METHOD RaiseSyncUnitEvent
VAR_INPUT
	EventId	  : UDINT;
	Argument1 : STRING := '';
	Argument2 : STRING := '';
	Argument3 : STRING := '';
END_VAR
IF Argument3 <> '' THEN
	SyncUnitEvents.Arguments(EventId).Clear().AddString(Argument1).AddString(Argument2).AddString(Argument3);
ELSIF Argument2 <> '' THEN
	SyncUnitEvents.Arguments(EventId).Clear().AddString(Argument1).AddString(Argument2);
ELSIF Argument1 <> '' THEN
	SyncUnitEvents.Arguments(EventId).Clear().AddString(Argument1);
ELSE
	SyncUnitEvents.Arguments(EventId).Clear();
END_IF

SyncUnitEvents.RaiseEvent(EventId);
END_METHOD

METHOD Reset
SyncUnitEvents.Reset();
EtherCatMasterEvents.Reset();
END_METHOD

METHOD SetEventReactions
VAR_INPUT
	Verbose	 : DINT := 0;
	Info	 : DINT := 1;
	Warning	 : DINT := 2;
	Error	 : DINT := 3;
	Critical : DINT := 4;
END_VAR
SyncUnitEvents.SetEventReactions(Verbose,
								 Info,
								 Warning,
								 Error,
								 Critical);

EtherCatMasterEvents.SetEventReactions(Verbose,
									   Info,
									   Warning,
									   Error,
									   Critical);
END_METHOD

(*FB_Init is always available implicitly and it is used primarily for initialization.
The return value is not evaluated. For a specific influence, you can also declare the
methods explicitly and provide additional code there with the standard initialization
code. You can evaluate the return value.*)
METHOD FB_Init : BOOL
VAR_INPUT
	(* TRUE: the retain variables are initialized (reset warm / reset cold)*)
	bInitRetains : BOOL;

	(* TRUE: the instance will be copied to the copy code afterward (online change)   *)
	bInCopyCode				 : BOOL;
	Name					 : Core.T_MaxString;
	EtherCatMasterDiagnostic : I_EtherCatMasterDiagnostic;
END_VAR
THIS^.EtherCatMasterDiagnostic := EtherCatMasterDiagnostic;
THIS^.EtherCatMasterDiagnostic.RegisterEventProvider(THIS^);
SyncUnitEvents.GenerateTcEvents(EtherCatMasterDiagnostic.Name, ADR(TC_Events.SyncUnit), SIZEOF(ST_SyncUnit));
EtherCatMasterEvents.GenerateTcEvents(EtherCatMasterDiagnostic.Name, ADR(TC_Events.EtherCatMaster), SIZEOF(ST_EtherCatMaster));
END_METHOD

END_FUNCTION_BLOCK

// Components/Recipe/Interface/I_RecipeManagment
INTERFACE I_RecipeManagment EXTENDS I_Component

{attribute 'monitoring' := 'call'}
PROPERTY AutoLoadChangesToActive : BOOL
SET
END_SET
END_PROPERTY

{attribute 'monitoring' := 'call'}
PROPERTY ChangesPending : BOOL
GET
END_GET
END_PROPERTY

METHOD LoadChangesToActive
VAR_INPUT
END_VAR
END_METHOD

END_INTERFACE

// Components/Recipe/RecipeManagment
FUNCTION_BLOCK RecipeManagment EXTENDS CyclicComponent IMPLEMENTS I_RecipeManagment
VAR
	nRecipe					 : UDINT;
	pActiveRecipeData		 : PVOID;
	pUpdateRecipeData		 : PVOID;
	_ChangesPending			 : BOOL;
	_AutoLoadChangesToActive : BOOL;
END_VAR

METHOD CyclicLogic
IF nRecipe = 0 THEN
	RETURN;
END_IF

IF pActiveRecipeData = 0 THEN
	RETURN;
END_IF

IF pUpdateRecipeData = 0 THEN
	RETURN;
END_IF

CompareData();
END_METHOD

METHOD CompareData
VAR_INPUT
END_VAR
IF MEMCMP(pActiveRecipeData, pUpdateRecipeData, nRecipe) = 0 THEN
	_ChangesPending := FALSE;
ELSE
	IF _AutoLoadChangesToActive THEN
		LoadChangesToActive();
	ELSE
		_ChangesPending := TRUE;
	END_IF
END_IF
END_METHOD

{attribute 'monitoring' := 'call'}
PROPERTY AutoLoadChangesToActive : BOOL
SET
_AutoLoadChangesToActive := AutoLoadChangesToActive;
END_SET
END_PROPERTY

{attribute 'monitoring' := 'call'}
PROPERTY ChangesPending : BOOL
GET
ChangesPending := _ChangesPending;
END_GET
END_PROPERTY

METHOD LoadChangesToActive
VAR_INPUT
END_VAR
MEMCPY(pActiveRecipeData, pUpdateRecipeData, nRecipe);
CompareData();
END_METHOD

(*FB_Init is always available implicitly and it is used primarily for initialization.
The return value is not evaluated. For a specific influence, you can also declare the
methods explicitly and provide additional code there with the standard initialization
code. You can evaluate the return value.*)
METHOD FB_Init : BOOL
VAR_INPUT
	(* TRUE: the retain variables are initialized (reset warm / reset cold)*)
	bInitRetains : BOOL;

	(* TRUE: the instance will be copied to the copy code afterward (online change)   *)
	bInCopyCode		  : BOOL;
	Name			  : Core.T_MaxString;
	nRecipe			  : UDINT;
	pActiveRecipeData : PVOID;
	pUpdateRecipeData : PVOID;
END_VAR
THIS^.nRecipe			:= nRecipe;
THIS^.pActiveRecipeData := pActiveRecipeData;
THIS^.pUpdateRecipeData := pUpdateRecipeData;
END_METHOD

END_FUNCTION_BLOCK

// Components/Safety/Interface/I_InSafetyGroup
INTERFACE I_InSafetyGroup EXTENDS I_Base

PROPERTY SafetyGroup : I_TaskResult
SET
END_SET
END_PROPERTY

END_INTERFACE

// Components/Safety/Interface/I_SafetyBase
INTERFACE I_SafetyBase EXTENDS I_Component, I_Resettable, I_SafetySimulation, I_TaskResult

{attribute 'monitoring' := 'call'}
PROPERTY OK : BOOL
GET
END_GET
END_PROPERTY

PROPERTY ResetFunction : I_SafetyReset
SET
END_SET
END_PROPERTY

END_INTERFACE

// Components/Safety/Interface/I_SafetySimulation
INTERFACE I_SafetySimulation EXTENDS I_Simulatable

METHOD SimulateSafetyDiag
VAR_INPUT
	SimulationValueDiag : UINT;
END_VAR
END_METHOD

METHOD SimulateSafetyState
VAR_INPUT
	SimulationValueState : USINT;
END_VAR
END_METHOD

END_INTERFACE

// Components/Safety/Interface/I_SafetyReset
INTERFACE I_SafetyReset EXTENDS I_Cyclic, I_TaskResult

METHOD Execute
VAR_INPUT
END_VAR
END_METHOD

PROPERTY PulseDuration : TIME
SET
END_SET
END_PROPERTY

END_INTERFACE

// Components/Safety/Interface/I_SafetyModule
INTERFACE I_SafetyModule EXTENDS I_SafetySimulation, I_TaskResult, I_Resettable, I_Module

METHOD AddSafetyComponent
VAR_INPUT
	Component : I_SafetyBase;
END_VAR
END_METHOD

{attribute 'monitoring' := 'call'}
PROPERTY OK : BOOL
GET
END_GET
END_PROPERTY

PROPERTY SafetyPlcCoE : I_CoeDevice
GET
END_GET
END_PROPERTY

END_INTERFACE

// Components/Safety/Reset Function/SafetyResetPulse
FUNCTION_BLOCK SafetyResetPulse EXTENDS CyclicComponent IMPLEMENTS I_SafetyReset
VAR
	Reset AT %Q*   : BOOL;
	TpErrorAck	   : TP;
	TofErrorAck	   : TOF;
	_PulseDuration : TIME := T#100MS;
	_Error		   : BOOL;
	_Busy		   : BOOL;
END_VAR

METHOD CyclicLogic
TpErrorAck(PT := _PulseDuration, Q => Reset);
IF TpErrorAck.Q THEN
	TpErrorAck.IN := FALSE;
END_IF

TofErrorAck(In := TpErrorAck.Q, PT := _PulseDuration);
_Error := FALSE;
_Busy  := TofErrorAck.Q;
END_METHOD

{attribute 'monitoring' := 'call'}
PROPERTY Busy : BOOL
GET
Busy := _Busy;
END_GET
END_PROPERTY

{attribute 'monitoring' := 'call'}
PROPERTY Error : BOOL
GET
Error := _Error;
END_GET
END_PROPERTY

{attribute 'monitoring' := 'call'}
PROPERTY ErrorId : UDINT
GET
END_GET
END_PROPERTY

METHOD Execute
IF TpErrorAck.Q THEN
	RETURN;
END_IF

TpErrorAck.IN := TRUE;
END_METHOD

PROPERTY PulseDuration : TIME
SET
_PulseDuration := PulseDuration;
END_SET
END_PROPERTY

END_FUNCTION_BLOCK

// Components/Safety/Visitor/SafetyOkVisitor
FUNCTION_BLOCK SafetyOkVisitor IMPLEMENTS I_ComponentVisitor
VAR
	{attribute 'hide'}
	_OK				: BOOL;
	SafetyComponent : I_SafetyBase;
	ErrorComponent	: Core.I_Component;
END_VAR

{attribute 'monitoring' := 'call'}
PROPERTY OK : BOOL
GET
OK := _OK;
END_GET
END_PROPERTY

METHOD VisitComponent
VAR_INPUT
	Component : Core.I_Component;
END_VAR
_OK := TRUE;
IF __QUERYINTERFACE(Component, SafetyComponent) THEN
	IF NOT SafetyComponent.OK THEN
		ErrorComponent := Component;
		_OK			   := FALSE;
	END_IF
END_IF
END_METHOD

END_FUNCTION_BLOCK

// Components/Safety/Visitor/SetSafetySimulationVisitor
FUNCTION_BLOCK SetSafetySimulationVisitor IMPLEMENTS I_ComponentVisitor
VAR
	SafetyComponent : I_SafetyBase;
	InfoData		: ST_SafetyStateDiag;
	_Simulated		: BOOL;
END_VAR

PROPERTY Diag : UINT
SET
InfoData.Diag := Diag;
END_SET
END_PROPERTY

PROPERTY Simulated : BOOL
GET
Simulated := _Simulated;
END_GET
SET
_Simulated := Simulated;
END_SET
END_PROPERTY

PROPERTY State : USINT
SET
InfoData.State := State;
END_SET
END_PROPERTY

METHOD VisitComponent
VAR_INPUT
	Component : Core.I_Component;
END_VAR
IF __QUERYINTERFACE(Component, SafetyComponent) THEN
	SafetyComponent.Simulated := _Simulated;
	SafetyComponent.SimulateSafetyDiag(InfoData.Diag);
	SafetyComponent.SimulateSafetyState(InfoData.State);
END_IF
END_METHOD

END_FUNCTION_BLOCK

// Components/Safety/SafetyAndOrFB
FUNCTION_BLOCK SafetyAndOrFB EXTENDS SafetyBase
VAR
END_VAR

METHOD CyclicLogic
VAR_INST
	LinkError : BOOL;
END_VAR
SUPER^.CyclicLogic();
_OK := SUPER^.InfoData.State = E_SafetyOrAnd_State.Run;
END_METHOD

END_FUNCTION_BLOCK

// Components/Safety/SafetyBase
FUNCTION_BLOCK SafetyBase EXTENDS CyclicComponent IMPLEMENTS I_SafetyBase
VAR
	InfoData AT %I* : ST_SafetyStateDiag;
	{attribute 'hide'}
	_Simulated : BOOL;
	{attribute 'hide'}
	_OK : BOOL;
	{attribute 'hide'}
	_Error : BOOL;
	{attribute 'hide'}
	_Busy : BOOL;
	{attribute 'hide'}
	_ErrorId	   : UDINT;
	_ResetFunction : I_SafetyReset;
END_VAR

METHOD CyclicLogic
VAR_INST
	LinkError : BOOL;
END_VAR
IF NOT LinkError AND NOT Simulated AND (F_GetMappingStatus(ADR(InfoData), SIZEOF(InfoData)) = EplcMappingStatus.MS_Unmapped) THEN
	LinkError := TRUE;
	Trace.LogMessage(Name, 'Not mapped to Safety, no diagnostics available!');
END_IF

IF _ResetFunction <> 0 THEN
	_ResetFunction.CyclicLogic();
END_IF
END_METHOD

{attribute 'monitoring' := 'call'}
PROPERTY OK : BOOL
GET
OK := _OK;
END_GET
END_PROPERTY

METHOD Reset
IF _ResetFunction <> 0 THEN
	_ResetFunction.Execute();
END_IF
END_METHOD

PROPERTY ResetFunction : I_SafetyReset
SET
_ResetFunction := ResetFunction;
END_SET
END_PROPERTY

{attribute 'monitoring' := 'call'}
PROPERTY Simulated : BOOL
GET
Simulated := _Simulated;
END_GET
SET
_Simulated := Simulated;
END_SET
END_PROPERTY

METHOD SimulateSafetyDiag
VAR_INPUT
	SimulationValueDiag : UINT;
END_VAR
Infodata.Diag := SimulationValueDiag;
END_METHOD

METHOD SimulateSafetyState
VAR_INPUT
	SimulationValueState : USINT;
END_VAR
Infodata.State := SimulationValueState;
END_METHOD

{attribute 'monitoring' := 'call'}
PROPERTY Busy : BOOL
GET
Busy := _Busy;
END_GET
END_PROPERTY

{attribute 'monitoring' := 'call'}
PROPERTY Error : BOOL
GET
Error := _Error;
END_GET
END_PROPERTY

{attribute 'monitoring' := 'call'}
PROPERTY ErrorId : UDINT
GET
ErrorId := _ErrorId;
END_GET
END_PROPERTY

END_FUNCTION_BLOCK

// Components/Safety/SafetyConnectionFB_TcEvents
FUNCTION_BLOCK SafetyConnectionFB_TcEvents EXTENDS SafetyBase IMPLEMENTS I_EventReactionTcEvents
VAR
	Events : TcEventClass('FSoE Connection Events');
END_VAR

METHOD CyclicLogic
VAR_INST
	DiagWord	: WORD;
	BitMaskDiag : WORD := 16#000F;
END_VAR
SUPER^.CyclicLogic();
_OK	   := SUPER^.InfoData.State = E_SafetyConnection_State.Data;
_Error := GetHighestActiveEventReaction() >= TcEventSeverity.Error;
IF _ResetFunction <> 0 AND_THEN _ResetFunction.Busy THEN
	RETURN;
END_IF

BitMaskDiag := 16#000F;
DiagWord	:= TO_WORD(SUPER^.InfoData.Diag) AND BitMaskDiag;
IF (DiagWord = 1) THEN
	Events.RaiseEvent(E_SafetyConnection.InvalidCommand);
END_IF

IF (DiagWord = 2) THEN
	Events.RaiseEvent(E_SafetyConnection.UnknownCommand);
END_IF

IF (DiagWord = 3) THEN
	Events.RaiseEvent(E_SafetyConnection.InvalidConID);
END_IF

IF (DiagWord = 4) THEN
	Events.RaiseEvent(E_SafetyConnection.InvalidCrc);
END_IF

IF (DiagWord = 5) THEN
	Events.RaiseEvent(E_SafetyConnection.WatchdogExpired);
END_IF

IF (DiagWord = 6) THEN
	Events.RaiseEvent(E_SafetyConnection.InvalidFSOEAddr);
END_IF

IF (DiagWord = 7) THEN
	Events.RaiseEvent(E_SafetyConnection.InvalidData);
END_IF

IF (DiagWord = 8) THEN
	Events.RaiseEvent(E_SafetyConnection.InvalidComParameterLen);
END_IF

IF (DiagWord = 9) THEN
	Events.RaiseEvent(E_SafetyConnection.InavlidComParameter);
END_IF

IF (DiagWord = 10) THEN
	Events.RaiseEvent(E_SafetyConnection.InvalidUserParameterLen);
END_IF

IF (DiagWord = 11) THEN
	Events.RaiseEvent(E_SafetyConnection.InvalidUserParameter);
END_IF

IF (DiagWord = 12) THEN
	Events.RaiseEvent(E_SafetyConnection.FSoEMasterReset);
END_IF

IF (DiagWord = 13) THEN
	Events.RaiseEvent(E_SafetyConnection.ModuleErrorOnSlave);
END_IF

IF (DiagWord = 14) THEN
	Events.RaiseEvent(E_SafetyConnection.ModuleError);
END_IF

IF (DiagWord = 15) THEN
	Events.RaiseEvent(E_SafetyConnection.SlaveNotStarted);
END_IF

BitMaskDiag := 16#0010;
DiagWord	:= TO_WORD(SUPER^.InfoData.Diag) AND BitMaskDiag;
IF DiagWord.4 THEN
	Events.RaiseEvent(E_SafetyConnection.FsoESlaveError);
END_IF

BitMaskDiag := 16#0020;
DiagWord	:= TO_WORD(SUPER^.InfoData.Diag) AND BitMaskDiag;
IF DiagWord.5 THEN
	Events.RaiseEvent(E_SafetyConnection.FsoESlaveFailSafeValue);
END_IF

BitMaskDiag := 16#0040;
DiagWord	:= TO_WORD(SUPER^.InfoData.Diag) AND BitMaskDiag;
IF DiagWord.6 THEN
	Events.RaiseEvent(E_SafetyConnection.Startup);
END_IF

BitMaskDiag := 16#0080;
DiagWord	:= TO_WORD(SUPER^.InfoData.Diag) AND BitMaskDiag;
IF DiagWord.7 THEN
	Events.RaiseEvent(E_SafetyConnection.FsoEMasterSafeValue);
END_IF

IF SUPER^.InfoData.Diag.3 THEN
	Events.RaiseEvent(E_SafetyEstop.Disc4);
END_IF

IF SUPER^.InfoData.Diag.4 THEN
	Events.RaiseEvent(E_SafetyEstop.EDM1);
END_IF

IF SUPER^.InfoData.Diag.5 THEN
	Events.RaiseEvent(E_SafetyEstop.EDM2);
END_IF
END_METHOD

METHOD GetHighestActiveEventReaction : DINT
GetHighestActiveEventReaction := Events.GetHighestActiveEventReaction();
END_METHOD

METHOD GetHighestActiveEventSeverity : Core.TcEventSeverity
GetHighestActiveEventSeverity := Events.GetHighestActiveEventSeverity();
END_METHOD

METHOD Reset
SUPER^.Reset();
Events.Reset();
END_METHOD

METHOD SetEventReactions
VAR_INPUT
	Verbose	 : DINT := 0;
	Info	 : DINT := 1;
	Warning	 : DINT := 2;
	Error	 : DINT := 3;
	Critical : DINT := 4;
END_VAR
Events.SetEventReactions(Verbose,
						 Info,
						 Warning,
						 Error,
						 Critical);
END_METHOD

(*FB_Init is always available implicitly and it is used primarily for initialization.
The return value is not evaluated. For a specific influence, you can also declare the
methods explicitly and provide additional code there with the standard initialization
code. You can evaluate the return value.*)
METHOD FB_Init : BOOL
VAR_INPUT
	(* TRUE: the retain variables are initialized (reset warm / reset cold)*)
	bInitRetains : BOOL;

	(* TRUE: the instance will be copied to the copy code afterward (online change)   *)
	bInCopyCode : BOOL;
	Name		: Core.T_MaxString;
END_VAR
Events.GenerateTcEvents(Name, ADR(TC_events.SafetyConnection), SIZEOF(ST_SafetyConnection));
END_METHOD

END_FUNCTION_BLOCK

// Components/Safety/SafetyEdmFB_TcEvents
FUNCTION_BLOCK SafetyEdmFB_TcEvents EXTENDS SafetyBase IMPLEMENTS I_EventReactionTcEvents, I_InSafetyGroup
VAR
	Events		 : TcEventClass('Safety EDM Events');
	_SafetyGroup : I_TaskResult;
END_VAR

METHOD CyclicLogic
SUPER^.CyclicLogic();
_OK	   := SUPER^.InfoData.State <> E_SafetyEdm_State.Error;
_Error := GetHighestActiveEventReaction() >= TcEventSeverity.Error;
IF _SafetyGroup <> 0 THEN
	IF _SafetyGroup.Error THEN
		Events.Reset();
		RETURN;
	END_IF
END_IF

IF _ResetFunction <> 0 AND_THEN _ResetFunction.Busy THEN
	RETURN;
END_IF

IF SUPER^.InfoData.Diag.0 THEN
	Events.RaiseEvent(E_SafetyEdm.SwitchOffTime);
END_IF

IF SUPER^.InfoData.Diag.1 THEN
	Events.RaiseEvent(E_SafetyEdm.SwitchOnTime);
END_IF
END_METHOD

METHOD GetHighestActiveEventReaction : DINT
GetHighestActiveEventReaction := Events.GetHighestActiveEventReaction();
END_METHOD

METHOD GetHighestActiveEventSeverity : Core.TcEventSeverity
GetHighestActiveEventSeverity := Events.GetHighestActiveEventSeverity();
END_METHOD

METHOD Reset
SUPER^.Reset();
Events.Reset();
END_METHOD

METHOD SetEventReactions
VAR_INPUT
	Verbose	 : DINT := 0;
	Info	 : DINT := 1;
	Warning	 : DINT := 2;
	Error	 : DINT := 3;
	Critical : DINT := 4;
END_VAR
Events.SetEventReactions(Verbose,
						 Info,
						 Warning,
						 Error,
						 Critical);
END_METHOD

(*FB_Init is always available implicitly and it is used primarily for initialization.
The return value is not evaluated. For a specific influence, you can also declare the
methods explicitly and provide additional code there with the standard initialization
code. You can evaluate the return value.*)
METHOD FB_Init : BOOL
VAR_INPUT
	(* TRUE: the retain variables are initialized (reset warm / reset cold)*)
	bInitRetains : BOOL;

	(* TRUE: the instance will be copied to the copy code afterward (online change)   *)
	bInCopyCode : BOOL;
	Name		: Core.T_MaxString;
END_VAR
Events.GenerateTcEvents(Name, ADR(TC_events.SafetyEdm), SIZEOF(ST_SafetyEdm));
END_METHOD

PROPERTY SafetyGroup : I_TaskResult
SET
_SafetyGroup := SafetyGroup;
END_SET
END_PROPERTY

END_FUNCTION_BLOCK

// Components/Safety/SafetyEstopFB_TcEvents
FUNCTION_BLOCK SafetyEstopFB_TcEvents EXTENDS SafetyBase IMPLEMENTS I_EventReactionTcEvents, I_InSafetyGroup
VAR
	{attribute 'hide'}
	_ActiveName	 : STRING := 'pressed!';
	Events		 : TcEventClass('Safety E-Stop Events');
	_SafetyGroup : I_TaskResult;
END_VAR

METHOD CyclicLogic
SUPER^.CyclicLogic();
_OK	   := SUPER^.InfoData.State = E_SafetyEStop_State.Run;
_Error := GetHighestActiveEventReaction() >= TcEventSeverity.Error;
IF _SafetyGroup <> 0 THEN
	IF _SafetyGroup.Error THEN
		Events.Reset();
		RETURN;
	END_IF
END_IF

IF _ResetFunction <> 0 AND_THEN _ResetFunction.Busy THEN
	RETURN;
END_IF

IF NOT SUPER^.OK THEN
	Events.Arguments(E_SafetyEstop.Active).Clear().AddString(_ActiveName);
	Events.RaiseEvent(E_SafetyEstop.Active);
END_IF

IF SUPER^.InfoData.Diag.0 THEN
	Events.RaiseEvent(E_SafetyEstop.Disc1);
END_IF

IF SUPER^.InfoData.Diag.1 THEN
	Events.RaiseEvent(E_SafetyEstop.Disc2);
END_IF

IF SUPER^.InfoData.Diag.2 THEN
	Events.RaiseEvent(E_SafetyEstop.Disc3);
END_IF

IF SUPER^.InfoData.Diag.3 THEN
	Events.RaiseEvent(E_SafetyEstop.Disc4);
END_IF

IF SUPER^.InfoData.Diag.4 THEN
	Events.RaiseEvent(E_SafetyEstop.EDM1);
END_IF

IF SUPER^.InfoData.Diag.5 THEN
	Events.RaiseEvent(E_SafetyEstop.EDM2);
END_IF
END_METHOD

METHOD GetHighestActiveEventReaction : DINT
GetHighestActiveEventReaction := Events.GetHighestActiveEventReaction();
END_METHOD

METHOD GetHighestActiveEventSeverity : Core.TcEventSeverity
GetHighestActiveEventSeverity := Events.GetHighestActiveEventSeverity();
END_METHOD

METHOD Reset
SUPER^.Reset();
Events.Reset();
END_METHOD

METHOD SetEventReactions
VAR_INPUT
	Verbose	 : DINT := 0;
	Info	 : DINT := 1;
	Warning	 : DINT := 2;
	Error	 : DINT := 3;
	Critical : DINT := 4;
END_VAR
Events.SetEventReactions(Verbose,
						 Info,
						 Warning,
						 Error,
						 Critical);
END_METHOD

{attribute 'monitoring' := 'call'}
PROPERTY ActiveName : STRING
SET
_ActiveName := ActiveName;
END_SET
END_PROPERTY

(*FB_Init is always available implicitly and it is used primarily for initialization.
The return value is not evaluated. For a specific influence, you can also declare the
methods explicitly and provide additional code there with the standard initialization
code. You can evaluate the return value.*)
METHOD FB_Init : BOOL
VAR_INPUT
	(* TRUE: the retain variables are initialized (reset warm / reset cold)*)
	bInitRetains : BOOL;

	(* TRUE: the instance will be copied to the copy code afterward (online change)   *)
	bInCopyCode : BOOL;
	Name		: Core.T_MaxString;
END_VAR
Events.GenerateTcEvents(Name, ADR(TC_events.SafetyEstop), SIZEOF(ST_SafetyEstop));
END_METHOD

PROPERTY SafetyGroup : I_TaskResult
SET
_SafetyGroup := SafetyGroup;
END_SET
END_PROPERTY

END_FUNCTION_BLOCK

// Components/Safety/SafetyGroup_TcEvents
FUNCTION_BLOCK SafetyGroup_TcEvents EXTENDS SafetyBase IMPLEMENTS I_EventReactionTcEvents
VAR
	Run AT %Q* : BOOL;
	Events	   : TcEventClass('Safety Group Events');
	{attribute 'hide'}
	_AutoResetFaults : BOOL;
END_VAR

METHOD CyclicLogic
VAR_INST
	LinkErrorRun	 : BOOL;
	AutoFaultAck	 : TON;
	TriggerAutoReset : R_TRIG;
END_VAR
SUPER^.CyclicLogic();
IF NOT LinkErrorRun AND NOT Simulated AND (F_GetMappingStatus(ADR(Run), SIZEOF(Run)) = EplcMappingStatus.MS_Unmapped) THEN
	LinkErrorRun := TRUE;
	Trace.LogMessage(Name, 'Group Run not mapped to Safety!');
END_IF

Run := TRUE;
IF _ResetFunction <> 0 THEN
	AutoFaultAck(IN := (_AutoResetFaults AND (SUPER^.InfoData.Diag <> 0)) AND NOT _ResetFunction.Busy, PT := T#250MS);
	TriggerAutoReset(CLK := AutoFaultAck.Q);
	IF TriggerAutoReset.Q THEN
		_ResetFunction.Execute();
	END_IF

	_Busy := _ResetFunction.Busy;
END_IF

_OK	   := SUPER^.InfoData.State = E_SafetyGroup_State.Run;
_Error := GetHighestActiveEventReaction() >= TcEventSeverity.Error;
IF _ResetFunction <> 0 AND_THEN _ResetFunction.Busy THEN
	RETURN;
END_IF

IF SUPER^.InfoData.Diag = E_SafetyGroup_Diag.FbError THEN
	Events.RaiseEvent(E_SafetyGroup.FbError);
END_IF

IF SUPER^.InfoData.Diag = E_SafetyGroup_Diag.ComError THEN
	Events.RaiseEvent(E_SafetyGroup.ComError);
END_IF

IF SUPER^.InfoData.Diag = E_SafetyGroup_Diag.ModuleError THEN
	Events.RaiseEvent(E_SafetyGroup.ModuleError);
END_IF

IF SUPER^.InfoData.Diag = E_SafetyGroup_Diag.CmpError THEN
	Events.RaiseEvent(E_SafetyGroup.ModuleError);
END_IF

IF SUPER^.InfoData.Diag = E_SafetyGroup_Diag.DeactiveError THEN
	Events.RaiseEvent(E_SafetyGroup.DeactiveError);
END_IF

IF SUPER^.InfoData.Diag = E_SafetyGroup_Diag.RestartError THEN
	Events.RaiseEvent(E_SafetyGroup.RestartError);
END_IF
END_METHOD

METHOD GetHighestActiveEventReaction : DINT
GetHighestActiveEventReaction := Events.GetHighestActiveEventReaction();
END_METHOD

METHOD GetHighestActiveEventSeverity : Core.TcEventSeverity
GetHighestActiveEventSeverity := Events.GetHighestActiveEventSeverity();
END_METHOD

METHOD Reset
SUPER^.Reset();
Events.Reset();
END_METHOD

METHOD SetEventReactions
VAR_INPUT
	Verbose	 : DINT := 0;
	Info	 : DINT := 1;
	Warning	 : DINT := 2;
	Error	 : DINT := 3;
	Critical : DINT := 4;
END_VAR
Events.SetEventReactions(Verbose,
						 Info,
						 Warning,
						 Error,
						 Critical);
END_METHOD

{attribute 'monitoring' := 'call'}
PROPERTY AutoResetFaults : BOOL
GET
AutoResetFaults := _AutoResetFaults;
END_GET
SET
_AutoResetFaults := AutoResetFaults;
END_SET
END_PROPERTY

(*FB_Init is always available implicitly and it is used primarily for initialization.
The return value is not evaluated. For a specific influence, you can also declare the
methods explicitly and provide additional code there with the standard initialization
code. You can evaluate the return value.*)
METHOD FB_Init : BOOL
VAR_INPUT
	(* TRUE: the retain variables are initialized (reset warm / reset cold)*)
	bInitRetains : BOOL;

	(* TRUE: the instance will be copied to the copy code afterward (online change)   *)
	bInCopyCode : BOOL;
	Name		: Core.T_MaxString;
END_VAR
Events.GenerateTcEvents(Name, ADR(TC_events.SafetyGroup), SIZEOF(ST_SafetyGroup));
END_METHOD

END_FUNCTION_BLOCK

// Components/Safety/SafetyModule
FUNCTION_BLOCK SafetyModule EXTENDS Module IMPLEMENTS I_SafetyModule
VAR
	SequenceState			 : UDINT;
	TwinSAFEResetDelay		 : TON;
	SafetyPLC_WcState AT %I* : BOOL;
	SafetyPLC_AmsAddr AT %I* : AMSADDR;
	_SafetyPlcCoE			 : CoeDevice('Safety PLC') := (AdsAddr := SafetyPLC_AmsAddr);
	_SafetyAddressInfo		 : ST_SafetyAddressInfo;
END_VAR

VAR
	GetComponentsTaskResultVisitor : GetComponentsTaskResultVisitor;
	SetSafetySimulationVisitor	   : SetSafetySimulationVisitor;
	SafetyOkVisitor				   : SafetyOkVisitor;
END_VAR

METHOD OnCyclicCall
IF NOT Initialized THEN
	Initialize();
	RETURN;
END_IF

TwinSAFEResetDelay(PT := T#250MS);
CASE SequenceState OF
	0:
		TwinSAFEResetDelay.IN := FALSE;

	10:
		ResetComponents();
		SequenceState := 20;

	20:
		TwinSAFEResetDelay.IN := TRUE;
		IF TwinSAFEResetDelay.Q THEN
			SequenceState := 0;
		END_IF
END_CASE

GetComponentsTaskResultVisitor.Update(THIS^);
THIS^.Components.Accept(SafetyOkVisitor);
END_METHOD

(* This Module will be done initialize when ModuleInitialized := TRUE;, subequently all subitems will be called to be initialized *)
METHOD Initializing
_SafetyPlcCoE.CyclicLogic();
CASE SequenceState OF
	0:
		IF F_GetMappingStatus(ADR(SafetyPLC_WcState), SIZEOF(SafetyPLC_WcState)) = EplcMappingStatus.MS_Unmapped OR F_GetMappingStatus(ADR(SafetyPLC_AmsAddr), SIZEOF(SafetyPLC_AmsAddr)) = EplcMappingStatus.MS_Unmapped THEN
			SequenceState := 100;
			Trace.LogMessage(Name, 'Safety PLC not mapped, info will not be read!');
		ELSE
			SequenceState := SequenceState + 10;
		END_IF

	10:
		IF NOT SafetyPLC_WcState THEN
			SequenceState := SequenceState + 10;
		END_IF

	20:
		SafetyPlcCoE.Read(16#F980,
						  1,
						  ADR(_SafetyAddressInfo.FSoEAddress),
						  SIZEOF(_SafetyAddressInfo.FSoEAddress));

		SequenceState := SequenceState + 1;

	21:
		IF NOT SafetyPlcCoE.Error AND NOT SafetyPlcCoE.Busy THEN
			SequenceState := SequenceState + 1;
		END_IF

	22:
		SafetyPlcCoE.Read(16#F980,
						  2,
						  ADR(_SafetyAddressInfo.SerialNumber),
						  SIZEOF(_SafetyAddressInfo.SerialNumber));

		SequenceState := SequenceState + 1;

	23:
		IF NOT SafetyPlcCoE.Error AND NOT SafetyPlcCoE.Busy THEN
			SequenceState := SequenceState + 1;
		END_IF

	24:
		SafetyPlcCoE.Read(16#F980,
						  3,
						  ADR(_SafetyAddressInfo.ProjectCRC),
						  SIZEOF(_SafetyAddressInfo.ProjectCRC));

		SequenceState := SequenceState + 1;

	25:
		IF NOT SafetyPlcCoE.Error AND NOT SafetyPlcCoE.Busy THEN
			SequenceState := SequenceState + 1;
		END_IF

	26:
		SafetyPlcCoE.Read(16#F980,
						  4,
						  ADR(_SafetyAddressInfo.DefaultProjectCRC),
						  SIZEOF(_SafetyAddressInfo.DefaultProjectCRC));

		SequenceState := SequenceState + 1;

	27:
		IF NOT SafetyPlcCoE.Error AND NOT SafetyPlcCoE.Busy THEN
			SequenceState := 100;
		END_IF

	100:
		SequenceState	  := 0;
		ModuleInitialized := TRUE;
END_CASE
END_METHOD

{attribute 'monitoring' := 'call'}
PROPERTY Simulated : BOOL
GET
Simulated := SetSafetySimulationVisitor.Simulated;
END_GET
SET
SetSafetySimulationVisitor.Simulated := Simulated;
Components.Accept(SetSafetySimulationVisitor);
END_SET
END_PROPERTY

METHOD SimulateSafetyDiag
VAR_INPUT
	SimulationValueDiag : UINT;
END_VAR
SetSafetySimulationVisitor.Diag := SimulationValueDiag;
Components.Accept(SetSafetySimulationVisitor);
END_METHOD

METHOD SimulateSafetyState
VAR_INPUT
	SimulationValueState : USINT;
END_VAR
SetSafetySimulationVisitor.State := SimulationValueState;
Components.Accept(SetSafetySimulationVisitor);
END_METHOD

{attribute 'monitoring' := 'call'}
PROPERTY Busy : BOOL
GET
Busy := SequenceState <> 0;
END_GET
END_PROPERTY

{attribute 'monitoring' := 'call'}
PROPERTY Error : BOOL
GET
Error := GetComponentsTaskResultVisitor.Error;
END_GET
END_PROPERTY

{attribute 'monitoring' := 'call'}
PROPERTY ErrorId : UDINT
GET
ErrorId := GetComponentsTaskResultVisitor.ErrorId;
END_GET
END_PROPERTY

METHOD AddSafetyComponent
VAR_INPUT
	Component : I_SafetyBase;
END_VAR
Component.RegisterWithParent(THIS^);
END_METHOD

(*FB_Init is always available implicitly and it is used primarily for initialization.
The return value is not evaluated. For a specific influence, you can also declare the
methods explicitly and provide additional code there with the standard initialization
code. You can evaluate the return value.*)
METHOD FB_Init : BOOL
VAR_INPUT
	(* TRUE: the retain variables are initialized (reset warm / reset cold)*)
	bInitRetains : BOOL;

	(* TRUE: the instance will be copied to the copy code afterward (online change)   *)
	bInCopyCode : BOOL;
	Name		: Core.T_MaxString;
END_VAR
SafetyPlcCoE.RegisterWithParent(THIS^);
END_METHOD

{attribute 'monitoring' := 'call'}
PROPERTY OK : BOOL
GET
OK := SafetyOkVisitor.OK;
END_GET
END_PROPERTY

METHOD Reset
IF Busy THEN
	RETURN;
END_IF

SequenceState := 10;
END_METHOD

PROPERTY SafetyAddressInfo : REFERENCE TO ST_SafetyAddressInfo
GET
SafetyAddressInfo REF= _SafetyAddressInfo;
END_GET
END_PROPERTY

PROPERTY SafetyPlcCoE : I_CoeDevice
GET
SafetyPlcCoE := _SafetyPlcCoE;
END_GET
END_PROPERTY

END_FUNCTION_BLOCK

// Components/Safety/SafetyMonFB_TcEvents
FUNCTION_BLOCK SafetyMonFB_TcEvents EXTENDS SafetyBase IMPLEMENTS I_EventReactionTcEvents, I_InSafetyGroup
VAR
	{attribute 'hide'}
	_ActiveAlarm : BOOL := TRUE;
	{attribute 'hide'}
	_ActiveName	 : STRING := 'pressed!';
	Events		 : TcEventClass('Safety MonFB Events');
	_SafetyGroup : I_TaskResult;
END_VAR

METHOD CyclicLogic
SUPER^.CyclicLogic();
_OK	   := SUPER^.InfoData.State = E_SafetyEStop_State.Run;
_Error := GetHighestActiveEventReaction() >= TcEventSeverity.Error;
IF _SafetyGroup <> 0 THEN
	IF _SafetyGroup.Error THEN
		Events.Reset();
		RETURN;
	END_IF
END_IF

IF _ResetFunction <> 0 AND_THEN _ResetFunction.Busy THEN
	RETURN;
END_IF

IF NOT SUPER^.OK AND _ActiveAlarm THEN
	Events.Arguments(E_SafetyMon.Active).Clear().AddString(_ActiveName);
	Events.RaiseEvent(E_SafetyMon.Active);
END_IF

IF SUPER^.InfoData.Diag.0 THEN
	Events.RaiseEvent(E_SafetyMon.Disc1);
END_IF

IF SUPER^.InfoData.Diag.1 THEN
	Events.RaiseEvent(E_SafetyMon.Disc2);
END_IF

IF SUPER^.InfoData.Diag.3 THEN
	Events.RaiseEvent(E_SafetyMon.DiscInput);
END_IF

IF SUPER^.InfoData.Diag.4 THEN
	Events.RaiseEvent(E_SafetyMon.Edm1);
END_IF

IF SUPER^.InfoData.Diag.5 THEN
	Events.RaiseEvent(E_SafetyMon.Edm2);
END_IF

IF SUPER^.InfoData.Diag.8 THEN
	Events.RaiseEvent(E_SafetyMon.Disc1Safe);
END_IF

IF SUPER^.InfoData.Diag.9 THEN
	Events.RaiseEvent(E_SafetyMon.Disc2Safe);
END_IF

IF SUPER^.InfoData.Diag.10 THEN
	Events.RaiseEvent(E_SafetyMon.DiscInputSafe);
END_IF
END_METHOD

METHOD GetHighestActiveEventReaction : DINT
GetHighestActiveEventReaction := Events.GetHighestActiveEventReaction();
END_METHOD

METHOD GetHighestActiveEventSeverity : Core.TcEventSeverity
GetHighestActiveEventSeverity := Events.GetHighestActiveEventSeverity();
END_METHOD

METHOD Reset
SUPER^.Reset();
Events.Reset();
END_METHOD

METHOD SetEventReactions
VAR_INPUT
	Verbose	 : DINT := 0;
	Info	 : DINT := 1;
	Warning	 : DINT := 2;
	Error	 : DINT := 3;
	Critical : DINT := 4;
END_VAR
Events.SetEventReactions(Verbose,
						 Info,
						 Warning,
						 Error,
						 Critical);
END_METHOD

PROPERTY ActiveAlarm : BOOL
SET
_ActiveAlarm := ActiveAlarm;
END_SET
END_PROPERTY

PROPERTY ActiveName : STRING
SET
_ActiveName := ActiveName;
END_SET
END_PROPERTY

(*FB_Init is always available implicitly and it is used primarily for initialization.
The return value is not evaluated. For a specific influence, you can also declare the
methods explicitly and provide additional code there with the standard initialization
code. You can evaluate the return value.*)
METHOD FB_Init : BOOL
VAR_INPUT
	(* TRUE: the retain variables are initialized (reset warm / reset cold)*)
	bInitRetains : BOOL;

	(* TRUE: the instance will be copied to the copy code afterward (online change)   *)
	bInCopyCode : BOOL;
	Name		: Core.T_MaxString;
END_VAR
Events.GenerateTcEvents(Name, ADR(TC_events.SafetyMon), SIZEOF(ST_SafetyMon));
END_METHOD

PROPERTY SafetyGroup : I_TaskResult
SET
_SafetyGroup := SafetyGroup;
END_SET
END_PROPERTY

END_FUNCTION_BLOCK

// Components/Tcp Ip/Interface/I_TcpIpConnection
INTERFACE I_TcpIpConnection EXTENDS I_Component

{attribute 'monitoring' := 'call'}
PROPERTY IP : T_IPv4Addr
SET
END_SET
END_PROPERTY

{attribute 'monitoring' := 'call'}
PROPERTY Port : UDINT
SET
END_SET
END_PROPERTY

METHOD RegisterCommand
VAR_INPUT
	Command : I_TcpIpSubscription;
END_VAR
END_METHOD

METHOD SendCommand
VAR_INPUT
	Command : STRING(4096);
END_VAR
END_METHOD

METHOD SendPriorityCommand
VAR_INPUT
	Command : STRING(4096);
END_VAR
END_METHOD

END_INTERFACE

// Components/Tcp Ip/Interface/I_TcpIpSubscription
INTERFACE I_TcpIpSubscription EXTENDS I_Base

METHOD UpdateCommandResult
VAR_INPUT
	Response : STRING(4096);
END_VAR
END_METHOD

END_INTERFACE

// Components/Tcp Ip/TcpIpCommandResultFilter
FUNCTION_BLOCK ABSTRACT TcpIpCommandResultFilter EXTENDS CyclicComponent IMPLEMENTS I_TcpIpSubscription
VAR
	TcpIpConnection : I_TcpIpConnection;
	{attribute 'hide'}
	_Initialized   : BOOL := FALSE;
	CommandActive  : BOOL;
	CommandTimeout : TON;

	//
	Response	  : STRING(4096);
	Command		  : STRING(4096);
	JsonSaxWriter : FB_JsonSaxWriter;
	JsonDocument  : SJsonValue;
	JsonValue	  : SJsonValue;
	JsonDomParser : FB_JsonDomParser;
END_VAR

METHOD CyclicLogic
CommandTimeout(IN := CommandActive, PT := T#10S);
IF CommandTimeout.Q THEN
	CommandActive := FALSE;
	Trace.Info(_Name, CONCAT('Command response not recieved! ', Name));
END_IF
END_METHOD

(*FB_Init is always available implicitly and it is used primarily for initialization.
The return value is not evaluated. For a specific influence, you can also declare the
methods explicitly and provide additional code there with the standard initialization
code. You can evaluate the return value.*)
METHOD FB_Init : BOOL
VAR_INPUT
	(* TRUE: the retain variables are initialized (reset warm / reset cold)*)
	bInitRetains : BOOL;

	(* TRUE: the instance will be copied to the copy code afterward (online change)   *)
	bInCopyCode		: BOOL;
	Name			: Core.T_MaxString;
	TcpIpConnection : I_TcpIpConnection;
END_VAR
THIS^.TcpIpConnection := TcpIpConnection;
TcpIpConnection.RegisterCommand(THIS^);
END_METHOD

METHOD ABSTRACT UpdateCommandResult
VAR_INPUT
	Response : STRING(4096);
END_VAR
// Filter incoming TcpIp traffic here!
END_METHOD

END_FUNCTION_BLOCK

// Components/Tcp Ip/TcpIpConnection
FUNCTION_BLOCK TcpIpConnection EXTENDS CyclicComponent IMPLEMENTS I_TcpIpConnection, I_Initializable
VAR
	_Initialized   : BOOL;
	_IP			   : T_IPv4Addr := '127.0.0.1';
	_Port		   : UDINT;
	SocketCloseAll : FB_SocketCloseAll;

	// Send Port
	ReconnectTimer		   : TON;
	ClientServerConnection : FB_ClientServerConnection;
	ServerConnectionState  : E_SocketConnectionState;
	SocketSend			   : FB_SocketSend;
	SendMessage			   : STRING(4096);
	Socket				   : T_HSOCKET;
	SendDelay			   : TON := (PT := T#100MS);
	PollTimer			   : TON;
	ResponseTimer		   : TON;
	SocketReceive		   : FB_SocketReceive;
	ReceiveMessage		   : STRING(4096);
END_VAR

VAR
	Commands		   : ARRAY[0..COMMAND_BUFFER] OF I_TcpIpSubscription;
	SendBuffer		   : ARRAY[0..COMMAND_BUFFER] OF STRING(4096);
	PrioritySendBuffer : ARRAY[0..COMMAND_BUFFER] OF STRING(4096);
END_VAR

VAR CONSTANT
	RECON_TIME	   : TIME := T#10S;
	COMMAND_BUFFER : DINT := 99;
END_VAR

METHOD CyclicLogic
IF NOT _Initialized THEN
	Initialize();
	RETURN;
END_IF

SendReceiveSequence();
END_METHOD

METHOD Initialize
SocketCloseAll(sSrvNetId := '', bExecute := TRUE);
IF NOT SocketCloseAll.bBusy AND NOT SocketCloseAll.bError THEN
	_Initialized := TRUE;
END_IF
END_METHOD

{attribute 'monitoring' := 'call'}
PROPERTY Initialized : BOOL
GET
Initialized := _Initialized;
END_GET
SET
_Initialized := Initialized;
END_SET
END_PROPERTY

METHOD PROTECTED EvaluateResponse
VAR
	i : DINT;
END_VAR
FOR i := 0 TO COMMAND_BUFFER DO
	IF Commands[i] = 0 THEN
		EXIT;
	END_IF

	Commands[i].UpdateCommandResult(ReceiveMessage);
END_FOR

MEMSET(ADR(ReceiveMessage), 0, SIZEOF(ReceiveMessage));
END_METHOD

METHOD PROTECTED GetNextCommand
VAR
	i : DINT;
END_VAR
IF SendBuffer[0] <> '' THEN
	SendMessage := SendBuffer[0];
	FOR i := 0 TO (COMMAND_BUFFER - 1) DO
		SendBuffer[i] := SendBuffer[i + 1];
	END_FOR
END_IF
END_METHOD

METHOD PROTECTED GetNextPriorityCommand
VAR
	i : DINT;
END_VAR
IF PrioritySendBuffer[0] <> '' THEN
	SendMessage := PrioritySendBuffer[0];
	FOR i := 0 TO (COMMAND_BUFFER - 1) DO
		PrioritySendBuffer[i] := PrioritySendBuffer[i + 1];
	END_FOR
END_IF
END_METHOD

METHOD PROTECTED SendReceiveSequence
VAR_INST
	SequenceState : UDINT;
END_VAR
ClientServerConnection(sSrvNetID   := '',
					   sRemoteHost := _IP,
					   nRemotePort := _Port,
					   hSocket	   => Socket,
					   eState	   => ServerConnectionState);

SocketSend(sSrvNetId := '',
		   hSocket	 := Socket,
		   cbLen	 := TO_UDINT(LEN(SendMessage)),
		   pSrc		 := ADR(SendMessage),
		   tTimeout	 := T#5S);

SocketReceive(sSrvNetId := '',
			  hSocket	:= Socket,
			  cbLen		:= SIZEOF(ReceiveMessage),
			  pDest		:= ADR(ReceiveMessage),
			  tTimeout	:= T#5S);

//
ReconnectTimer(PT := RECON_TIME);
PollTimer(PT := T#100MS);
ResponseTimer(PT := T#50S);
CASE SequenceState OF
	0:
		ClientServerConnection.bEnable := TRUE;
		IF ServerConnectionState = eSOCKET_CONNECTED THEN
			SequenceState := SequenceState + 10;
		END_IF

		IF ClientServerConnection.bError THEN
			Trace.Error(_Name, CONCAT('ClientServerConnection.bError: ', TO_STRING(ClientServerConnection.nErrId)));
			SequenceState := 200;
		END_IF

	10:
		// SENDING -----------------------------------------------------------------------------------
		SendDelay(IN := NOT SendDelay.Q);
		IF SendMessage = '' THEN
			GetNextPriorityCommand();
		END_IF

		IF SendMessage = '' THEN
			GetNextCommand();
		END_IF

		IF SocketSend.bExecute AND NOT SocketSend.bBusy AND NOT SocketSend.bError THEN
			Trace.Info(_Name, CONCAT('Client sent: ', SendMessage));
			MEMSET(ADR(SendMessage), 0, SIZEOF(SendMessage));
			SocketSend.bExecute := FALSE;
		END_IF

		IF SendMessage <> '' AND NOT SocketSend.bExecute AND SendDelay.Q THEN
			SocketSend.bExecute := TRUE;
		END_IF

		IF SocketSend.bError THEN
			Trace.Error(_Name, CONCAT('SocketSend.bError: ', TO_STRING(SocketSend.nErrId)));
			SequenceState := 200;
		END_IF

		// RECEIVING -----------------------------------------------------------------------------------
		PollTimer.IN		   := TRUE;
		SocketReceive.bExecute := TRUE;
		IF PollTimer.Q AND NOT SocketReceive.bError AND NOT SocketReceive.bBusy THEN
			IF SocketReceive.nRecBytes > 0 THEN
				ResponseTimer.IN := FALSE;
				Trace.Info(_Name, CONCAT('Client recieved: ', ReceiveMessage));
				EvaluateResponse();
			END_IF

			SequenceState := 11;
			// Stale connection, disconnected while socket was open
			IF SocketReceive.nRecBytes = 0 THEN
				ResponseTimer.IN := TRUE;
				IF ResponseTimer.Q THEN
					Trace.Error(_Name, 'Receive Connection stale - re-connect!');
					SequenceState := 200;
				END_IF
			END_IF
		END_IF

		IF SocketReceive.bError THEN
			Trace.Error(_Name, CONCAT('SocketReceive.bError: ', TO_STRING(SocketReceive.nErrId)));
			SequenceState := 200;
		END_IF

	11:
		PollTimer.IN		   := FALSE;
		SocketReceive.bExecute := FALSE;
		SequenceState		   := 10;

	200:
		ReconnectTimer.IN			   := TRUE;
		ResponseTimer.IN			   := FALSE;
		ClientServerConnection.bEnable := FALSE;
		SocketReceive.bExecute		   := FALSE;
		SocketSend.bExecute			   := FALSE;
		IF ServerConnectionState = eSOCKET_DISCONNECTED AND ReconnectTimer.Q THEN
			ReconnectTimer.IN := FALSE;
			SequenceState	  := 0;
		END_IF
END_CASE
END_METHOD

{attribute 'monitoring' := 'call'}
PROPERTY IP : T_IPv4Addr
SET
_IP := IP;
END_SET
END_PROPERTY

{attribute 'monitoring' := 'call'}
PROPERTY Port : UDINT
SET
_Port := Port;
END_SET
END_PROPERTY

METHOD RegisterCommand
VAR_INPUT
	Command : I_TcpIpSubscription;
END_VAR

VAR
	i : DINT;
END_VAR
FOR i := 0 TO COMMAND_BUFFER DO
	IF Commands[i] = 0 THEN
		Commands[i] := Command;
		RETURN;
	END_IF
END_FOR
END_METHOD

METHOD SendCommand
VAR_INPUT
	Command : STRING(4096);
END_VAR

VAR
	i : DINT;
END_VAR
FOR i := 0 TO COMMAND_BUFFER DO
	IF SendBuffer[i] = '' THEN
		SendBuffer[i] := Command;
		RETURN;
	END_IF
END_FOR
END_METHOD

METHOD SendPriorityCommand
VAR_INPUT
	Command : STRING(4096);
END_VAR

VAR
	i : DINT;
END_VAR
FOR i := 0 TO COMMAND_BUFFER DO
	IF PrioritySendBuffer[i] = '' THEN
		PrioritySendBuffer[i] := Command;
		RETURN;
	END_IF
END_FOR
END_METHOD

END_FUNCTION_BLOCK

// Project Information/F_GetCompany
// This function has been automatically generated from the project information.
{attribute 'signature_flag' := '1073741824'}
{attribute 'TcGenerated'}
{attribute 'no-analysis'}
FUNCTION F_GetCompany : WSTRING
VAR_INPUT
	
END_VAR

F_GetCompany := "Beckhoff Automation LLC";

END_FUNCTION

// Project Information/F_GetTitle
// This function has been automatically generated from the project information.
{attribute 'signature_flag' := '1073741824'}
{attribute 'TcGenerated'}
{attribute 'no-analysis'}
FUNCTION F_GetTitle : WSTRING
VAR_INPUT
	
END_VAR

F_GetTitle := "CoreComponents";

END_FUNCTION

// Project Information/F_GetVersion
// This function has been automatically generated from the project information.
{attribute 'signature_flag' := '1073741824'}
{attribute 'TcGenerated'}
{attribute 'no-analysis'}
FUNCTION F_GetVersion : ST_LibVersion
VAR_INPUT
	
END_VAR

F_GetVersion.iMajor := 1;
F_GetVersion.iMinor := 2;
F_GetVersion.iBuild := 2;
F_GetVersion.iRevision := 0;
F_GetVersion.sVersion := '1.2.2';
F_GetVersion.nFlags := 0;

END_FUNCTION

// Utilities/AnyBuffer/Interface/I_AnyBuffer
INTERFACE I_AnyBuffer

// Clears all buffer data and resets metadata to initial state
METHOD Clear : BOOL
END_METHOD

PROPERTY Configuration : REFERENCE TO ST_BufferConfiguration
GET
END_GET
END_PROPERTY

// Deletes element at specified index position and decrements element count
METHOD DeleteAtIndex : BOOL
VAR_INPUT
	index : DINT; // Zero-based index position of element to delete
END_VAR
END_METHOD

PROPERTY isEmpty : BOOL
GET
END_GET
END_PROPERTY

PROPERTY isFull : BOOL
GET
END_GET
END_PROPERTY

PROPERTY Metadata : REFERENCE TO ST_BufferMetadata
GET
END_GET
END_PROPERTY

// Retrieve an element at a specific index without removing it from the buffer
METHOD PeekAtIndex : BOOL
VAR_INPUT
	index	: DINT;
	element : ANY;
END_VAR
END_METHOD

// Remove and retrieve an element at a specific index, shifting remaining elements left
METHOD PopAtIndex : BOOL
VAR_INPUT
	index	   : DINT;
	element	   : ANY;
	popDiscard : BOOL := FALSE;
END_VAR
END_METHOD

// Removes and retrieves the first element from the buffer (FIFO/queue operation)
METHOD PopLeft : BOOL
VAR_INPUT
	element	   : ANY;			// Variable to receive the popped element
	popDiscard : BOOL := FALSE; // When TRUE, element is removed but not copied (type checking skipped)
END_VAR
END_METHOD

// Removes and retrieves the last element from the buffer (stack pop operation)
METHOD PopRight : BOOL
VAR_INPUT
	element	   : ANY;			// Variable to receive the popped element
	popDiscard : BOOL := FALSE; // When TRUE, element is removed but not copied (type checking skipped)
END_VAR
END_METHOD

// Add an element at a specific index, shifting remaining elements right
METHOD PushAtIndex : BOOL
VAR_INPUT
	index	: DINT;
	element : ANY;
END_VAR
END_METHOD

// Appends a new element to the left side of the buffer (LIFO/stack push operation)
METHOD PushLeft : BOOL
VAR_INPUT
	element : ANY;
END_VAR
END_METHOD

// Appends a new element to the right side of the buffer (FIFO/queue enqueue operation)
METHOD PushRight : BOOL
VAR_INPUT
	element : ANY;
END_VAR
END_METHOD

// Replaces an element at a specific index with the given element
METHOD ReplaceAtIndex : BOOL
VAR_INPUT
	index	: DINT;
	element : ANY;
END_VAR
END_METHOD

END_INTERFACE

// Utilities/AnyBuffer/Interface/I_AnyBufferStrategy
INTERFACE I_AnyBufferStrategy

METHOD Clear : BOOL
END_METHOD

PROPERTY isEmpty : BOOL
GET
END_GET
END_PROPERTY

PROPERTY isFull : BOOL
GET
END_GET
END_PROPERTY

END_INTERFACE

// Utilities/AnyBuffer/TypedBuffers/FifoBuffer
// Provides a simplified FIFO queue interface as an adapter over AnyBuffer
FUNCTION_BLOCK FifoBuffer IMPLEMENTS I_AnyBufferStrategy
VAR
	anyBuffer	  : I_AnyBuffer;
	isInitialized : BOOL := FALSE;
	_overwrite	  : BOOL := FALSE; // When TRUE, Push overwrites oldest element when full
	_reversed	  : BOOL := FALSE; // When TRUE, reverses push/pop direction (PushLeft/PopRight)
	{attribute 'hide'}
	discardObject : BYTE; // element for discarding elements in overwrite mode
END_VAR

(*
## Detailed Description

FifoBuffer is an adapter (also known as a strategy or facade) that wraps an AnyBuffer instance
to provide a simplified First-In-First-Out (FIFO) queue interface. Instead of using the full
AnyBuffer API with directional operations (AppendLeft/Right, PopLeft/Right), users can simply
Push and Pop elements following standard queue semantics.

### Alternative Names
In computer science, FIFO data structures are commonly called "Queues". This implementation
could alternatively be named "Queue" or "QueueAdapter" for more conventional naming.

### Design Pattern
This implements the **Adapter Pattern** (also Strategy Pattern), which:
- Wraps a more complex interface (I_AnyBuffer) with a simpler, domain-specific interface
- Delegates all operations to the underlying AnyBuffer instance
- Provides semantic clarity: Push/Pop vs AppendLeft/PopRight
- Allows multiple strategy implementations (FIFO, LIFO, Priority, etc.) over the same buffer

### FIFO Semantics
- **Push(element)**: Adds element using PushRight (reversed=FALSE) or PushLeft (reversed=TRUE)
- **Pop(element)**: Removes element using PopLeft (reversed=FALSE) or PopRight (reversed=TRUE)
- The reversed parameter controls the direction of both Push and Pop operations
- Elements maintain insertion order, but retrieval order depends on reversed setting

### Configurable Behavior
The FifoBuffer supports two optional parameters during initialization:

**overwrite parameter:**
- **FALSE (default)**: Push fails when buffer is full, returns FALSE and logs error
- **TRUE**: Push to full buffer automatically removes element to make space (circular buffer behavior)
  - When reversed=FALSE: Removes from front (PopLeft), adds to back (PushRight)
  - When reversed=TRUE: Removes from back (PopRight), adds to front (PushLeft)
  - Removed element is discarded using internal temporary buffer

**reversed parameter:**
- **FALSE (default)**: Standard FIFO - Push to back (PushRight), Pop from front (PopLeft)
- **TRUE**: Reversed direction - Push to front (PushLeft), Pop from back (PopRight)
- When reversed=TRUE, behavior is similar to LIFO/stack but with directional consistency

### Operation Mapping
**Standard Mode (overwrite=FALSE, reversed=FALSE):**
```
Push()  -> anyBuffer.PushRight()  // Add to back (right)
Pop()   -> anyBuffer.PopLeft()    // Remove from front (left)
Clear() -> anyBuffer.Clear()      // Clear all
isEmpty -> anyBuffer.isEmpty      // Check if empty
isFull  -> anyBuffer.isFull       // Check if full
```

**Overwrite Mode (overwrite=TRUE, reversed=FALSE):**
```
Push()  -> if full: anyBuffer.PopLeft(pBufferTemp), then anyBuffer.PushRight()
Pop()   -> anyBuffer.PopLeft()    // Remove from front (left)
```

**Reversed Mode (overwrite=FALSE, reversed=TRUE):**
```
Push()  -> anyBuffer.PushLeft()   // Add to front (left)
Pop()   -> anyBuffer.PopRight()   // Remove from back (right)
```

**Overwrite + Reversed Mode (overwrite=TRUE, reversed=TRUE):**
```
Push()  -> if full: anyBuffer.PopRight(pBufferTemp), then anyBuffer.PushLeft()
Pop()   -> anyBuffer.PopRight()   // Remove from back (right)
```

### Usage Examples

**Standard FIFO Mode:**
```iecst
VAR
    rawBuffer : ARRAY[0..2] OF DINT;
    buffer : AnyBuffer(pBuffer := rawBuffer,
                       bufferBoundLower := 0,
                       bufferBoundUpper := 2,
                       isBufferPersistent := FALSE);
    fifo : FifoBuffer(anyBuffer := buffer, overwrite := FALSE, reversed := FALSE);
    value : DINT;
END_VAR

// Push elements
value := 100; fifo.Push(value);  // Queue: [100]
value := 200; fifo.Push(value);  // Queue: [100, 200]
value := 300; fifo.Push(value);  // Queue: [100, 200, 300]

// Pop elements (FIFO order - oldest first)
fifo.Pop(value);   // value = 100, Queue: [200, 300]
fifo.Pop(value);   // value = 200, Queue: [300]
fifo.Pop(value);   // value = 300, Queue: []
```

**Overwrite Mode (Circular Buffer):**
```iecst
VAR
    fifo : FifoBuffer(anyBuffer := buffer, overwrite := TRUE, reversed := FALSE);
END_VAR

// Fill buffer
value := 100; fifo.Push(value);  // Queue: [100]
value := 200; fifo.Push(value);  // Queue: [100, 200]
value := 300; fifo.Push(value);  // Queue: [100, 200, 300]

// Push to full buffer overwrites oldest
value := 400; fifo.Push(value);  // Queue: [200, 300, 400] - 100 was removed
value := 500; fifo.Push(value);  // Queue: [300, 400, 500] - 200 was removed
```

**Reversed Mode (reversed=TRUE):**
```iecst
VAR
    fifo : FifoBuffer(anyBuffer := buffer, overwrite := FALSE, reversed := TRUE);
END_VAR

// Push elements (adds to front using PushLeft)
value := 100; fifo.Push(value);  // Buffer: [100]
value := 200; fifo.Push(value);  // Buffer: [200, 100] - 200 added to front
value := 300; fifo.Push(value);  // Buffer: [300, 200, 100] - 300 added to front

// Pop elements (removes from back using PopRight)
fifo.Pop(value);   // value = 100, Buffer: [300, 200]
fifo.Pop(value);   // value = 200, Buffer: [300]
fifo.Pop(value);   // value = 300, Buffer: []
```

### Advantages
- **Simplified interface**: Push/Pop instead of AppendLeft/PopRight
- **Semantic clarity**: Code intention is clearer with queue terminology
- **Flexibility**: Easy to swap different buffer strategies (FIFO, LIFO, etc.)
- **Type safety**: Enforces FIFO semantics at compile time through interface

### Limitations
- No random access: Cannot peek at arbitrary indices (use AnyBuffer directly if needed)
- No priority queue: Elements are strictly ordered by insertion time
- Overwrite mode loses oldest data when buffer is full
- Combining overwrite and reversed modes creates a circular stack behavior

### Dependencies
- Requires I_AnyBuffer implementation (e.g., AnyBuffer)
- Uses Trace for error logging and verbose diagnostics
- Implements I_AnyBufferStrategy interface

### Related Patterns
- **LifoBuffer**: Would implement stack (Last-In-First-Out) semantics
- **PriorityBuffer**: Would implement priority queue with ordered insertion
- **CircularBuffer**: Would implement ring buffer with overwrite semantics
*)

// Removes all elements from the queue and resets to empty state
METHOD Clear : BOOL

(*
## Detailed Description

Clears all elements from the underlying buffer, resetting it to an empty state.
After calling Clear, isEmpty will return TRUE and elementCount will be 0.

This operation delegates directly to the underlying anyBuffer.Clear() method.

### Return Value
- **TRUE**: Queue was successfully cleared
- **FALSE**: Clear operation failed (e.g., anyBuffer is not initialized)

### Side Effects
- All elements are removed from the buffer
- Element count is reset to 0
- Buffer capacity is restored to maximum
- Logs verbose trace message on success
*)
Clear := FALSE;
IF anyBuffer <> 0 THEN
	Clear := anyBuffer.Clear();
	;
END_IF

Trace.Verbose(__POUNAME(), 'executed');
END_METHOD

// Initializes the FIFO queue by injecting the underlying buffer dependency
METHOD FB_Init : BOOL
VAR_INPUT
	bInitRetains : BOOL;		// TRUE: the retain variables are initialized (reset warm / reset cold)
	bInCopyCode	 : BOOL;		// TRUE: the instance will be copied to the copy code afterward (online change)
	anyBuffer	 : I_AnyBuffer; // The underlying buffer implementation to wrap
	overwrite	 : BOOL;		// When TRUE, Push overwrites oldest element when full
	reversed	 : BOOL;		// When TRUE, reverses push/pop direction (PushLeft/PopRight)
END_VAR

(*
## Detailed Description

Initializes the FifoBuffer by injecting the underlying AnyBuffer dependency. This follows
the dependency injection pattern where the buffer implementation is provided during
construction rather than being created internally.

### Initialization Sequence
1. Validates that a valid anyBuffer reference is provided (non-zero pointer)
2. Stores the buffer reference for use by Push, Pop, and other operations
3. Sets isInitialized flag to TRUE to enable operations

### Parameters
- **anyBuffer**: Reference to an I_AnyBuffer implementation (e.g., AnyBuffer instance)
  - Must be a valid, initialized buffer
  - This FifoBuffer will delegate all operations to this buffer
- **overwrite**: Controls behavior when pushing to a full buffer
  - **FALSE (default)**: Push returns FALSE and logs error when buffer is full
  - **TRUE**: Push automatically removes an element to make space (circular buffer behavior)
    - When reversed=FALSE: Removes from front (PopLeft), adds to back (PushRight)
    - When reversed=TRUE: Removes from back (PopRight), adds to front (PushLeft)
  - Discarded element is popped to internal temporary buffer (pBufferTemp)
- **reversed**: Controls the direction of both Push and Pop operations
  - **FALSE (default)**: Push to back (PushRight), Pop from front (PopLeft) - standard FIFO
  - **TRUE**: Push to front (PushLeft), Pop from back (PopRight) - reversed direction
  - Affects the operational direction of the buffer, not just retrieval order

### Return Value
Returns BOOL but value is not evaluated by the runtime. Always call with valid anyBuffer.

### Usage Example
```iecst
VAR
    rawBuffer : ARRAY[0..9] OF DINT;
    buffer : AnyBuffer(pBuffer := rawBuffer,
                       bufferBoundLower := 0,
                       bufferBoundUpper := 9,
                       isBufferPersistent := FALSE);
    fifo : FifoBuffer(anyBuffer := buffer,
                      overwrite := FALSE,
                      reversed := FALSE);
END_VAR
```

### Important Notes
- Must provide a valid anyBuffer reference, otherwise Push/Pop will fail
- The underlying buffer must already be initialized before passing to FB_Init
- A temporary buffer (pBufferTemp) is allocated internally for discarding elements in overwrite mode
- pBufferTemp is automatically deallocated in FB_exit
- Overwrite mode is useful for logging/telemetry where newest data is more important
- Reversed mode changes the operational direction of both Push and Pop
- Combining overwrite=TRUE and reversed=TRUE creates a circular buffer operating from the opposite end
*)
IF anyBuffer <> 0 THEN
	THIS^.anyBuffer := anyBuffer;
	_overwrite		:= overwrite;
	_reversed		:= reversed;
	isInitialized	:= TRUE;
END_IF
END_METHOD

// Returns TRUE if the queue contains no elements
PROPERTY isEmpty : BOOL

(*
## Detailed Description

Returns TRUE if the queue is empty (contains no elements), FALSE otherwise.
This property delegates directly to the underlying anyBuffer.isEmpty property.

Use this property to check if Pop operation would succeed before attempting to
remove an element.

### Return Value
- **TRUE**: Queue is empty (elementCount = 0)
- **FALSE**: Queue contains one or more elements

### Usage Example
```iecst
IF NOT fifo.isEmpty THEN
    fifo.Pop(value);  // Safe to pop
END_IF
```
*)
GET
isEmpty := anyBuffer.isEmpty;
END_GET
END_PROPERTY

// Returns TRUE if the queue is at maximum capacity
PROPERTY isFull : BOOL

(*
## Detailed Description

Returns TRUE if the queue is full (at maximum capacity), FALSE otherwise.
This property delegates directly to the underlying anyBuffer.isFull property.

Use this property to check if Push operation would succeed before attempting to
add an element.

### Return Value
- **TRUE**: Queue is full (elementCount = capacity)
- **FALSE**: Queue has space for more elements

### Usage Example
```iecst
IF NOT fifo.isFull THEN
    value := 100;
    fifo.Push(value);  // Safe to push
END_IF
```
*)
GET
isFull := anyBuffer.isFull;
END_GET
END_PROPERTY

// Removes and retrieves an element from the queue (FIFO or LIFO depending on reversed setting)
{attribute 'hasanytype'}
METHOD Pop : BOOL
VAR_INPUT
	element : ANY; // Variable to receive the popped element
END_VAR

(*
## Detailed Description

Removes and retrieves an element from the queue. The behavior depends on the 'reversed'
initialization parameter:

**When reversed = FALSE (default mode):**
- Removes element from the front (left side, index 0)
- Delegates to anyBuffer.PopLeft()
- Standard FIFO behavior when combined with PushRight

**When reversed = TRUE (reversed mode):**
- Removes element from the back (right side, highest index)
- Delegates to anyBuffer.PopRight()
- Reversed direction - removes from opposite end compared to default
- Combined with PushLeft, maintains FIFO order but from opposite direction

### Operation Sequence
1. Validates that the buffer has been initialized
2. Validates that element size matches the buffer's configured element size
3. Checks that the queue is not empty
4. Removes element using PopLeft (FIFO) or PopRight (LIFO) based on reversed setting
5. Copies the element value to the output parameter
6. For PopLeft: Shifts remaining elements left; For PopRight: No shifting needed
7. Logs verbose trace on success or error trace on failure

### Standard Mode Example (reversed = FALSE)
```iecst
// Push to right, Pop from left
value := 100; fifo.Push(value);  // Buffer: [100]
value := 200; fifo.Push(value);  // Buffer: [100, 200] - 200 added to right
value := 300; fifo.Push(value);  // Buffer: [100, 200, 300] - 300 added to right

fifo.Pop(value);  // Returns 100 (from left), Buffer: [200, 300]
fifo.Pop(value);  // Returns 200 (from left), Buffer: [300]
fifo.Pop(value);  // Returns 300 (from left), Buffer: []
```

### Reversed Mode Example (reversed = TRUE)
```iecst
// Push to left, Pop from right
value := 100; fifo.Push(value);  // Buffer: [100]
value := 200; fifo.Push(value);  // Buffer: [200, 100] - 200 added to left
value := 300; fifo.Push(value);  // Buffer: [300, 200, 100] - 300 added to left

fifo.Pop(value);  // Returns 100 (from right), Buffer: [300, 200]
fifo.Pop(value);  // Returns 200 (from right), Buffer: [300]
fifo.Pop(value);  // Returns 300 (from right), Buffer: []
```

### Return Value
- **TRUE**: Element was successfully popped and copied to element parameter
- **FALSE**: Pop operation failed (see error conditions)

### Error Conditions
- Returns FALSE and logs error if buffer was not initialized
- Returns FALSE and logs error if element size doesn't match buffer element size
- Returns FALSE and logs error if queue is empty (no elements to pop)
- Returns FALSE and logs error if underlying PopLeft or PopRight operation fails

### Parameters
- **element**: Must be a writable variable (not a literal) of the correct size
  - Must match the buffer's configured element size
  - Will receive the popped element value on success

### Side Effects
- Removes one element from the queue
- Decrements element count by 1
- For FIFO mode (reversed=FALSE): Shifts remaining elements one position to the left
- For LIFO mode (reversed=TRUE): No element shifting required
- Logs verbose trace message on success
- Logs error trace message on failure
*)
Pop := FALSE;
IF NOT isInitialized THEN
	Trace.Error(__POUNAME(), 'Buffer was not initialized yet, execute method .init() at least once');
	RETURN;
END_IF

// valid sized element?
IF element.diSize <> anyBuffer.Configuration.elementSize THEN
	Trace.Error(__POUNAME(), 'Passed element to pop to is of improper size');
	RETURN;
END_IF

// retrieve element from buffer if there is any left
IF NOT isEmpty THEN
	IF _reversed THEN
		// LIFO mode: pop from back (newest first)
		Pop := anyBuffer.PopRight(element);
	ELSE
		// FIFO mode: pop from front (oldest first)
		Pop := anyBuffer.PopLeft(element);
	END_IF
ELSE
	Trace.Error(__POUNAME(), 'Attempt to pop from empty buffer');
END_IF

// Pop was ok, trace message
IF Pop THEN
	Trace.Verbose(__POUNAME(), 'executed');
ELSE
	Trace.Error(__POUNAME(), 'FAILED');
END_IF
END_METHOD

// Adds a new element to the queue (direction depends on reversed setting)
{attribute 'hasanytype'}
METHOD Push : BOOL
VAR_INPUT
	element : ANY; // Element to add to the queue
END_VAR

(*
## Detailed Description

Adds a new element to the queue. The push direction and overwrite behavior depend on
the 'reversed' and 'overwrite' initialization parameters.

**Push Direction (reversed parameter):**
- **reversed = FALSE (default)**: Delegates to anyBuffer.PushRight() - adds to back/right
- **reversed = TRUE**: Delegates to anyBuffer.PushLeft() - adds to front/left

**Overwrite Behavior (overwrite parameter):**
- **overwrite = FALSE (default)**: Push fails if buffer is full, returns FALSE and logs error
- **overwrite = TRUE (circular buffer mode)**: Push succeeds even when buffer is full
  - When reversed=FALSE: Removes element from front (PopLeft to pBufferTemp), then adds to back (PushRight)
  - When reversed=TRUE: Removes element from back (PopRight to pBufferTemp), then adds to front (PushLeft)
  - Discarded element is popped to internal temporary buffer and dropped
  - Useful for logging/telemetry where newest data is more important

### Operation Sequence

**Standard Mode (overwrite = FALSE, reversed = FALSE):**
1. Validates that the buffer has been initialized
2. Validates that element size matches the buffer's configured element size
3. Checks that the queue is not full (has available capacity)
4. If full: Returns FALSE and logs error
5. If not full: Adds element to the back using PushRight
6. Logs verbose trace on success or error trace on failure

**Standard Mode with Reversed (overwrite = FALSE, reversed = TRUE):**
1. Validates that the buffer has been initialized
2. Validates that element size matches the buffer's configured element size
3. Checks that the queue is not full (has available capacity)
4. If full: Returns FALSE and logs error
5. If not full: Adds element to the front using PushLeft
6. Logs verbose trace on success or error trace on failure

**Overwrite Mode (overwrite = TRUE, reversed = FALSE):**
1. Validates that the buffer has been initialized
2. Validates that element size matches the buffer's configured element size
3. If buffer is full: Removes oldest element using PopLeft (discards to pBufferTemp)
4. Adds new element to the back using PushRight
5. Logs verbose trace on success or error trace on failure

**Overwrite Mode with Reversed (overwrite = TRUE, reversed = TRUE):**
1. Validates that the buffer has been initialized
2. Validates that element size matches the buffer's configured element size
3. If buffer is full: Removes element using PopRight (discards to pBufferTemp)
4. Adds new element to the front using PushLeft
5. Logs verbose trace on success or error trace on failure

### Standard Mode Example (overwrite = FALSE)
```iecst
// Starting with empty queue
value := 100; fifo.Push(value);  // Queue: [100]
value := 200; fifo.Push(value);  // Queue: [100, 200]
value := 300; fifo.Push(value);  // Queue: [100, 200, 300]

// Pop operations retrieve in FIFO order (oldest first)
fifo.Pop(value);  // Returns 100 (first pushed)
fifo.Pop(value);  // Returns 200 (second pushed)
fifo.Pop(value);  // Returns 300 (third pushed)
```

### Overwrite Mode Example (overwrite = TRUE)
```iecst
// Assuming buffer capacity is 3
value := 100; fifo.Push(value);  // Queue: [100]
value := 200; fifo.Push(value);  // Queue: [100, 200]
value := 300; fifo.Push(value);  // Queue: [100, 200, 300] - full

// Push to full buffer overwrites oldest
value := 400; fifo.Push(value);  // Queue: [200, 300, 400] - 100 removed
value := 500; fifo.Push(value);  // Queue: [300, 400, 500] - 200 removed
```

### Return Value
- **TRUE**: Element was successfully pushed to the queue
- **FALSE**: Push operation failed (see error conditions)

### Error Conditions
- Returns FALSE and logs error if buffer was not initialized
- Returns FALSE and logs error if element size doesn't match buffer element size
- Returns FALSE and logs error if queue is full AND overwrite is FALSE
- Returns FALSE and logs error if underlying PushRight operation fails
- In overwrite mode, Push should always succeed unless buffer is not initialized or element size is wrong

### Parameters
- **element**: Must be a writable variable (not a literal) of the correct size
  - Must match the buffer's configured element size
  - Value will be copied into the queue

### Side Effects

**Standard Mode (overwrite = FALSE):**
- Adds one element to the queue at the back (next available index)
- No shifting of existing elements required
- Increments element count by 1
- Decrements available capacity by 1
- Logs verbose trace message on success
- Logs error trace message on failure

**Overwrite Mode (overwrite = TRUE):**
- If buffer is full: Removes oldest element first (PopLeft with shifting)
- Adds new element to the back (next available index)
- Element count remains constant when overwriting
- Logs verbose trace message on success
- Logs error trace message on failure

### Performance Considerations
- **Standard mode (reversed=FALSE)**: O(1) - PushRight is constant time, no shifting
- **Standard mode (reversed=TRUE)**: O(n) - PushLeft requires shifting all elements right
- **Overwrite mode (reversed=FALSE)**: O(n) when full (PopLeft + PushRight both with shifting)
- **Overwrite mode (reversed=TRUE)**: O(n) when full (PopRight O(1) + PushLeft O(n))
- **Overwrite mode**: O(1) or O(n) when not full (depends on reversed setting)
- Pop operation with reversed=FALSE has O(n) complexity (PopLeft with shifting)
- Pop operation with reversed=TRUE has O(1) complexity (PopRight, no shifting)
- Trade-off: reversed=FALSE optimizes Push, reversed=TRUE optimizes Pop
*)
Push := FALSE;
IF NOT isInitialized THEN
	Trace.Error(__POUNAME(), 'Buffer was not initialized yet, execute method .init() at least once');
	RETURN;
END_IF

// valid sized element pushed?
IF element.diSize <> anyBuffer.Configuration.elementSize THEN
	Trace.Error(__POUNAME(), 'Pushed element is of improper size');
	RETURN;
END_IF

// handle full buffer based on overwrite setting
IF isFull THEN
	IF _overwrite THEN
		// Overwrite mode: remove element to make space (discard to pBufferTemp)
		IF _reversed THEN
			// Reversed: remove from back before adding to front
			anyBuffer.PopRight(discardObject, TRUE);
		ELSE
			// Standard: remove from front before adding to back
			anyBuffer.PopLeft(discardObject, TRUE);
		END_IF
	ELSE
		// Standard mode: fail and log error
		Trace.Error(__POUNAME(), 'Attempt to push to full buffer');
		RETURN;
	END_IF
END_IF

// add element based on direction setting
IF _reversed THEN
	// Reversed: add to front (left)
	Push := anyBuffer.PushLeft(element);
ELSE
	// Standard: add to back (right)
	Push := anyBuffer.PushRight(element);
END_IF

// Push was ok, trace message
IF Push THEN
	Trace.Verbose(__POUNAME(), 'executed');
ELSE
	Trace.Error(__POUNAME(), 'FAILED');
END_IF
END_METHOD

END_FUNCTION_BLOCK

// Utilities/AnyBuffer/AnyBuffer
// the AnyBuffer block behaves as a double ended que

// elements can be appended / popped left and right
FUNCTION_BLOCK AnyBuffer IMPLEMENTS I_AnyBuffer
VAR
	bufferConfiguration : ST_BufferConfiguration;
	isInitialized		: BOOL := FALSE;
	pBuffer				: ANYTYPE;
	{attribute 'hide'}
	pBufferTemp : POINTER TO BYTE;
END_VAR

VAR PERSISTENT
	bufferMetadata : ST_BufferMetadata;
END_VAR

PROPERTY buffer : ANYTYPE
GET
buffer := pBuffer;
END_GET
END_PROPERTY

// Clears all buffer data and resets metadata to initial state
METHOD Clear : BOOL

(*
## Detailed Description

Clears all data from the buffer and resets the metadata to its initial state. This method
performs a complete buffer reset by zeroing out both the buffer contents and all tracking
metadata, effectively returning the buffer to an empty, initialized state.

### Operation Sequence
1. Validates that the buffer has been properly initialized via FB_init/Initialize
2. Clears all buffer data using memset (sets all bytes to 0x00)
3. Clears all metadata (elementCount, capacity, etc.) using memset
4. Logs success or failure via Trace system

### Key Features
- **Complete reset**: Zeros out both buffer data and metadata structures
- **Initialization check**: Validates buffer is initialized before attempting clear
- **Safe operation**: Cannot corrupt uninitialized or invalid buffers
- **Comprehensive logging**: Traces verbose success or error failure messages
- **Fast execution**: Uses memset for efficient memory clearing

### Usage Example
```iecst
VAR
    buffer : AnyBuffer(pBuffer := myArray, bufferBoundLower := 0, bufferBoundUpper := 9, isBufferPersistent := FALSE);
    success : BOOL;
END_VAR

// Add some data
buffer.PushRight(value1);
buffer.PushRight(value2);

// Clear all data
success := buffer.Clear();
IF success THEN
    // Buffer is now empty, elementCount = 0
    // All buffer positions are zeroed
END_IF
```

### Return Value
- **TRUE**: Buffer was successfully cleared (both data and metadata)
- **FALSE**: Clear operation failed (buffer not initialized)

### Error Conditions
- Returns FALSE and logs error if buffer was not properly initialized
- This prevents clearing invalid or uninitialized memory regions

### Side Effects
- Sets all buffer element positions to zero (0x00)
- Resets elementCount to 0
- Resets all other metadata fields to 0
- Buffer can be immediately reused after successful clear

### Dependencies
- Requires buffer to be initialized via FB_init or Initialize method
- Uses memset for memory clearing operations
- Uses Trace for logging (Verbose for success, Error for failure)

### Performance Considerations
- Time complexity: O(n) where n = total buffer size in bytes
- Memory operations: Two memset calls (buffer data + metadata structure)
- Fast operation: memset is highly optimized for bulk memory operations

### Unittests
 - ClearsAllElements : verify all buffer positions are zeroed after Clear
 - ResetsElementCount : verify elementCount is reset to 0 after Clear
 - ResetsAllMetadata : verify all metadata fields (elementCount, capacity, etc.) are zeroed
 - ReturnsTrue : verify Clear returns TRUE when buffer is initialized
 - ClearEmptyBuffer : verify clearing an already-empty buffer returns TRUE
 - ClearAfterPush : verify Clear works correctly after pushing elements
 - ClearAfterPop : verify Clear works correctly after popping elements
 - MultipleClearCalls : verify consecutive Clear calls all return TRUE
 - ClearFullBuffer : verify Clear works when buffer is at capacity
 - ClearPartialBuffer : verify Clear works when buffer is partially filled
 - PreservesConfiguration : verify buffer configuration (capacity, elementSize) unchanged after Clear
 - CanReuseAfterClear : verify buffer can be reused (push/pop) immediately after Clear
*)
Clear := FALSE;
IF isInitialized THEN
	// Clear the local buffer
	memset(pBuffer.pValue, 16#0, TO_UDINT(pBuffer.diSize));
	memset(ADR(BufferMetadata), 16#0, SIZEOF(BufferMetadata));

	// after bufferMetadata clear re-set capacity
	bufferMetadata.capacity := bufferConfiguration.capacity;
	Clear					:= TRUE;
ELSE
	Trace.Error(__POUNAME(), 'Buffer was not properly initialized before clearing buffer');
END_IF

IF Clear THEN
	Trace.Verbose(__POUNAME(), 'executed');
ELSE
	Trace.Error(__POUNAME(), 'FAILED');
END_IF
END_METHOD

PROPERTY Configuration : REFERENCE TO ST_BufferConfiguration
GET
Configuration REF= bufferConfiguration;
END_GET
END_PROPERTY

METHOD PRIVATE CountDecrement
// Decrement element count, increment capacity
bufferMetadata.elementCount := bufferMetadata.elementCount - 1;
bufferMetadata.capacity		:= bufferMetadata.capacity + 1;
END_METHOD

METHOD PRIVATE CountIncrement
// Increment element count, decrement capacity
bufferMetadata.elementCount := bufferMetadata.elementCount + 1;
bufferMetadata.capacity		:= bufferMetadata.capacity - 1;
END_METHOD

// Deletes element at specified index position, BUT DOES NOT SHIFT
METHOD DeleteAtIndex : BOOL
VAR_INPUT
	index : DINT;
END_VAR

VAR
	offset		 : DINT;
	destAddr	 : PVOID;
	srcAddr		 : PVOID;
	nBytes		 : UDINT;
	rebasedIndex : DINT;
END_VAR

(*
## Detailed Description

Deletes the element at the specified index position by zeroing out its memory location.
This is a low-level primitive operation that clears data in place without shifting other
elements or modifying metadata counters. The caller is responsible for managing element
count and buffer state if needed.

### Operation Sequence
1. Validates that index is within valid range [0, capacity)
2. Calculates byte offset to the target element position
3. Clears the element data using memset (sets all bytes to 0x00)
4. Returns TRUE on successful deletion

### Key Features
- **Low-level primitive**: Does NOT modify metadata counters - caller's responsibility
- **No state checking**: Does NOT validate if position is filled or if buffer is empty
- **Direct deletion**: Clears data at specific index WITHOUT shifting elements
- **Bounds checking**: Validates index against capacity only (not elementCount)
- **Memory safety**: Prevents deletion at invalid indices
- **Error logging**: Traces error with index value when deletion fails

### Usage Example
```iecst
VAR
    buffer : AnyBuffer(pBuffer := myArray, bufferBoundLower := 0, bufferBoundUpper := 9, isBufferPersistent := FALSE);
    success : BOOL;
END_VAR

// Delete element at index 3 (caller must manage elementCount)
success := buffer.DeleteAtIndex(3);
IF success THEN
    // Element at index 3 is now zeroed
    // NOTE: elementCount is NOT changed - caller must decrement if needed
END_IF
```

### Important Notes
- **No metadata changes**: Does NOT modify elementCount or any other metadata
- **Caller responsibility**: Calling code must manage element count if required
- **No shifting**: Does NOT shift remaining elements to fill the gap
- **No state checking**: Works regardless of whether position is filled or buffer is empty
- **Index range**: Valid indices are [0, capacity-1], not [0, elementCount-1]
- **Internal use**: Primarily used internally by PopLeft, PopRight, and PopAtIndex

### Return Value
- **TRUE**: Element was successfully deleted (zeroed at specified index)
- **FALSE**: Deletion failed due to invalid index (out of bounds)

### Error Conditions
- Returns FALSE and logs error if index < 0
- Returns FALSE and logs error if index >= capacity
- Error message includes the invalid index value for debugging

### Side Effects
- Zeros out all bytes of the element at the specified index
- **Does NOT** modify bufferMetadata.elementCount
- **Does NOT** modify any other element positions
- **Does NOT** shift elements to maintain contiguity
- **Does NOT** check if position was filled before deletion

### Dependencies
- Uses memset for memory clearing operation
- Uses Trace for error logging
- Requires valid buffer configuration (capacity, elementSize)

### Performance Considerations
- Time complexity: O(1) - constant time operation
- Memory operations: Single memset call for one element
- Fast operation: No element shifting, no metadata updates, no state checking

### Comparison with Other Methods
- **DeleteAtIndex**: Clears in place, no metadata change (O(1))
- **PopAtIndex**: Clears, shifts elements, updates count (O(n))
- **PopLeft/PopRight**: Specialized pop with shifting and count update (O(n))

### Unittests
 - DeletesAtValidIndex : verify element at valid index is zeroed after deletion
 - ReturnsTrueOnSuccess : verify method returns TRUE when deletion succeeds
 - ReturnsFalseOnInvalidIndex : verify method returns FALSE for out-of-bounds index
 - RejectsNegativeIndex : verify index < 0 is rejected with error log
 - RejectsIndexAtCapacity : verify index == capacity is rejected with error log
 - RejectsIndexAboveCapacity : verify index > capacity is rejected with error log
 - ExtremeBounds : verify rejection of extreme values like -10000 and very large positive indices
 - DeleteAtZero : verify deletion at first position (index 0) works correctly
 - DeleteAtCapacityMinusOne : verify deletion at last position (capacity-1) works correctly
 - DeleteAllPositions : verify deletion works correctly at all valid indices (0 through capacity-1)
 - PreservesOtherData : verify deletion at one index does not affect data at other indices
 - DeleteAlreadyEmpty : verify deleting an already-cleared position returns TRUE and remains zero
 - DeleteDoesNotShift : verify elements after deleted index remain at their original positions
 - DeleteWhenEmpty : verify deletion succeeds even when elementCount is 0 (clears position only)
 - MetadataUnchanged : verify elementCount and all metadata remain unchanged after deletion
 - ConsecutiveDeletesSamePosition : verify multiple deletes at same position succeed without metadata changes
*)
DeleteAtIndex := FALSE;
// check index
IF index < bufferConfiguration.bufferBoundLower OR index > bufferConfiguration.bufferBoundUpper THEN
	Trace.Error(__POUNAME(), CONCAT('Delete attempt at invalid index ', TO_STRING(index)));
	RETURN;
END_IF;

// rebasedIndex necessary if LL <> 0
rebasedIndex := index - bufferConfiguration.bufferBoundLower;

// Delete index element data
offset	 := rebasedIndex * bufferConfiguration.elementSize;
destAddr := ADR(pBuffer.pValue[offset]);
nBytes	 := TO_UDINT(bufferConfiguration.elementSize);
memset(destAddr, 16#0, nBytes);
DeleteAtIndex := TRUE;
END_METHOD

//FB_Exit must be implemented explicitly. If there is an implementation, then the

//method is called before the controller removes the code of the function block instance

//(implicit call). The return value is not evaluated.
METHOD FB_Exit : BOOL
VAR_INPUT
	bInCopyCode : BOOL; // TRUE: the exit method is called in order to leave the instance which will be copied afterwards (online change).  
END_VAR
__DELETE(pBufferTemp); // Delete if any exist
END_METHOD

//FB_Init is always available implicitly and it is used primarily for initialization.

//The return value is not evaluated. For a specific influence, you can also declare the

//methods explicitly and provide additional code there with the standard initialization

//code. You can evaluate the return value.
METHOD FB_Init : BOOL
VAR_INPUT
	bInitRetains	   : BOOL; // TRUE: the retain variables are initialized (reset warm / reset cold)
	bInCopyCode		   : BOOL; // TRUE: the instance will be copied to the copy code afterward (online change)   
	pBuffer			   : ANY;  // ANY to the buffer	
	bufferBoundLower   : DINT; // Lower boundary of the buffer
	bufferBoundUpper   : DINT; // Upper boundary of the buffer
	isBufferPersistent : BOOL; // Does the buffer need to be in persistent data?
END_VAR
THIS^.bufferConfiguration.isPersistent := isBufferPersistent;
// use the initialization method

// Valid pointer & strategy
IF pBuffer.pValue <> 0 THEN // AND_THEN
	//	bufferBoundLower = 0 			THEN
	THIS^.pBuffer						 := pBuffer;
	bufferConfiguration.bufferBoundLower := bufferBoundLower;
	bufferConfiguration.bufferBoundUpper := bufferBoundUpper;
	bufferConfiguration.capacity		 := bufferBoundUpper - bufferBoundLower + 1;
	IF NOT isBufferPersistent THEN
		// Clear the local buffer
		//memset(pBuffer.pValue, 16#0, TO_UDINT(pBuffer.diSize));
		memset(ADR(BufferMetadata), 16#0, SIZEOF(BufferMetadata));
	END_IF

	// At least 1 element? Is it an array?   	
	IF bufferConfiguration.capacity < 1 THEN
		// DO NOT USE TRACE IN THE FB_INIT METHODS
		// Trace.Error(__POUNAME(), 'Number of buffer elements < 1');
		bufferConfiguration.capacity := 0;
		isInitialized				 := FALSE;
	ELSE
		bufferConfiguration.elementSize := pBuffer.diSize / bufferConfiguration.capacity;
		bufferConfiguration.bufferSize	:= bufferConfiguration.capacity * bufferConfiguration.elementSize;
		IF NOT isBufferPersistent THEN
			// after bufferMetadata clear re-set capacity
			bufferMetadata.capacity := bufferConfiguration.capacity;
		END_IF

		// Temp buffer for the element
		pBufferTemp	  := __NEW(BYTE, TO_UDINT(bufferConfiguration.elementSize));
		isInitialized := TRUE;
	END_IF
END_IF
END_METHOD

METHOD FB_Reinit : BOOL
IF bufferConfiguration.elementSize > 0 THEN
	pBufferTemp := __NEW(BYTE, TO_UDINT(bufferConfiguration.elementSize));
END_IF
END_METHOD

PROPERTY isEmpty : BOOL
GET
isEmpty := (metaData.capacity >= bufferConfiguration.capacity);
END_GET
END_PROPERTY

PROPERTY isFull : BOOL
GET
isFull := (metaData.capacity <= 0);
END_GET
END_PROPERTY

PROPERTY Metadata : REFERENCE TO ST_BufferMetadata
GET
Metadata REF= bufferMetadata;
END_GET
END_PROPERTY

// Retrieve an element at a specific index without removing it from the buffer
METHOD PeekAtIndex : BOOL
VAR_INPUT
	index	: DINT;
	element : ANY;
END_VAR

VAR
	offset		 : DINT;
	destAddr	 : PVOID;
	srcAddr		 : PVOID;
	nBytes		 : UDINT;
	rebasedIndex : DINT;
END_VAR

(*
## Detailed Description

Retrieves an element at the specified index from the buffer without removing it or
modifying the buffer in any way. This is a read-only operation that provides random-access
read capability for the buffer. The buffer remains unchanged after this operation - no
elements are removed, shifted, or modified, and the element count stays the same.

### Operation Sequence
1. Validates that index is within valid range (0 to elementCount-1)
2. Validates that element size matches buffer element size (if element.diSize > 0)
3. Copies the element at the specified index to the output parameter
4. Returns without modifying the buffer

### Use Cases
```iecst
VAR
    buffer : AnyBuffer;
    value : DINT;
END_VAR

// Peek at elements without removing them
buffer.PushRight(100);  // [100]
buffer.PushRight(200);  // [100, 200]
buffer.PushRight(300);  // [100, 200, 300]

buffer.PeekAtIndex(0, value);  // value = 100, buffer still [100, 200, 300]
buffer.PeekAtIndex(1, value);  // value = 200, buffer still [100, 200, 300]
buffer.PeekAtIndex(2, value);  // value = 300, buffer still [100, 200, 300]

// Buffer unchanged - still contains all 3 elements
```

### Performance Considerations
- **Time complexity**: O(1) - constant time operation (direct indexed access)
- **Memory operations**: Single memcpy for element retrieval only
- **No buffer modifications**: No shifting, clearing, or count changes
- **Read-only**: Safe to call multiple times on same index
- Optimal for inspecting buffer contents without consumption
- Use for lookahead, validation, or monitoring buffer state

### Return Value
- **TRUE**: Element was successfully retrieved from the specified index
- **FALSE**: Peek operation failed (see error conditions)

### Error Conditions
- Returns FALSE and logs error if index is out of bounds (< 0 or >= elementCount)
- Returns FALSE and logs error if buffer is empty (elementCount = 0)
- Returns FALSE and logs error if element size doesn't match buffer element size (when element.diSize > 0)
- Element parameter can have diSize = 0 to skip copying (returns TRUE if index valid)

### Side Effects
- **None** - This is a read-only operation with no side effects
- Buffer contents remain unchanged
- Element count remains unchanged
- No elements are moved, cleared, or modified

### Dependencies
- Uses memcpy for element retrieval
- Uses Trace for error logging

### Comparison with Other Methods
- **PeekAtIndex**: Read element at any index - O(1), no modifications
- **PopAtIndex**: Read and remove element at any index - O(n), modifies buffer
- **PopLeft**: Read and remove first element - O(n), modifies buffer
- **PopRight**: Read and remove last element - O(1), modifies buffer
- **GetAtIndex** (if exists): Similar read-only operation

### Unittests
 - PeekFromBeginning : verify peeking at index 0 retrieves first element without modification
 - PeekFromMiddle : verify peeking from middle index retrieves correct element
 - PeekFromEnd : verify peeking at last index retrieves last element
 - ReturnsTrueOnSuccess : verify method returns TRUE when peek succeeds
 - ReturnsFalseOnNegativeIndex : verify FALSE returned for negative index
 - ReturnsFalseOnIndexOutOfBounds : verify FALSE returned when index >= elementCount
 - ReturnsFalseOnEmptyBuffer : verify FALSE returned when buffer is empty (elementCount = 0)
 - WrongElementSize : verify FALSE returned when element size doesn't match
 - EmptyElement : verify behavior when element.diSize is 0 (validation only, no copy)
 - BufferUnchangedAfterPeek : verify buffer contents unchanged after peek
 - ElementCountUnchanged : verify elementCount remains same after peek
 - MultiplePeeksOnSameIndex : verify can peek same index multiple times with consistent results
 - PeekAllPositions : verify can peek all valid positions in sequence
 - ElementOrderUnchanged : verify element order unchanged after multiple peeks
 - ConsecutivePeeks : verify multiple consecutive peeks at different indices work correctly
*)
PeekAtIndex := FALSE;
// Check index bounds, can peek every position even when not filled in
IF index < bufferConfiguration.bufferBoundLower OR index > bufferConfiguration.bufferBoundUpper THEN
	Trace.Error(__POUNAME(), CONCAT('Peek attempt at invalid index ', TO_STRING(index)));
	RETURN;
END_IF

// Check if buffer is empty
IF isEmpty THEN
	Trace.Error(__POUNAME(), 'Peek attempt on empty buffer');
	RETURN;
END_IF

// Check element size if copy is requested (element.diSize > 0)
IF element.diSize <> bufferConfiguration.elementSize THEN
	Trace.Error(__POUNAME(), CONCAT('Element size mismatch: expected ', CONCAT(TO_STRING(bufferConfiguration.elementSize), CONCAT(', got ', TO_STRING(element.diSize)))));
	RETURN;
END_IF

// rebasedIndex necessary if LL <> 0
rebasedIndex := index - bufferConfiguration.bufferBoundLower;

// Copy element at index to output parameter (if element.diSize > 0)
offset	 := rebasedIndex * bufferConfiguration.elementSize;
destAddr := element.pValue;
srcAddr	 := ADR(pBuffer.pValue[offset]);
nBytes	 := TO_UDINT(element.diSize);
memcpy(destAddr, srcAddr, nBytes);

// No buffer modifications - read-only operation
PeekAtIndex := TRUE;
END_METHOD

// Remove and retrieve an element at a specific index, decrement the element counter and shift remaining elements left
METHOD PopAtIndex : BOOL
VAR_INPUT
	index	   : DINT;
	element	   : ANY;
	popDiscard : BOOL := FALSE; // When TRUE, element is removed but not copied (type checking skipped)
END_VAR

VAR
	offset			: DINT;
	destAddr		: PVOID;
	srcAddr			: PVOID;
	nBytes			: UDINT;
	elementsToShift : DINT;
	rebasedIndex	: DINT;
END_VAR

(*
## Detailed Description

Removes an element at the specified index from the buffer and optionally copies it to
the provided element parameter. All elements after the removed index are shifted one
position to the left to maintain contiguous storage. This provides random-access pop
capability for the buffer, allowing removal from any position.

### Operation Sequence
1. Validates that index is within valid range (0 to elementCount-1)
2. Validates that element size matches buffer element size (if element.diSize > 0)
3. Copies the element at the specified index to the output parameter
4. Shifts all elements after the index one position to the left using MEMMOVE
5. Clears the last position (now empty after the shift)
6. Decrements the element count

### Use Cases
```iecst
VAR
    buffer : AnyBuffer;
    value : DINT;
END_VAR

// Remove element from middle of buffer
buffer.PushRight(100);  // [100]
buffer.PushRight(200);  // [100, 200]
buffer.PushRight(300);  // [100, 200, 300]
buffer.PopAtIndex(1, value);  // value = 200, buffer = [100, 300]
```

### Performance Considerations
- **Time complexity**: O(n) - requires shifting elements after the index
- **Memory operations**: One memcpy for retrieval, one MEMMOVE for shifting, one memset for clearing
- **Cost varies by index**:
  - PopAtIndex(0) is equivalent to PopLeft - shifts all remaining elements
  - PopAtIndex(elementCount-1) is equivalent to PopRight - no shifting needed
  - Middle indices require partial shifting
- Use PopRight for O(1) removal when index doesn't matter
- Use for priority queues or sorted list maintenance

### Return Value
- **TRUE**: Element was successfully popped from the specified index
- **FALSE**: Pop operation failed (see error conditions)

### Error Conditions
- Returns FALSE and logs error if index is out of bounds (< 0 or >= elementCount)
- Returns FALSE and logs error if buffer is empty (elementCount = 0)
- Returns FALSE and logs error if element size doesn't match buffer element size (when element.diSize > 0)
- Element parameter can have diSize = 0 to discard the value without copying

### Side Effects
- Shifts all elements after the index one position to the left
- Clears the last element position (sets to zero)
- Decrements bufferMetadata.elementCount by 1

### Dependencies
- Uses memcpy for element retrieval
- Uses MEMMOVE for shifting elements (handles overlapping memory)
- Uses memset for clearing the last position
- Uses Trace for error logging

### Comparison with Other Methods
- **PopAtIndex(0)**: Same as PopLeft - removes from front, shifts all - O(n)
- **PopAtIndex(elementCount-1)**: Same as PopRight - removes from back, no shift - O(1)
- **PopAtIndex(middle)**: Removes from middle, shifts elements after index - O(n)
- **DeleteAtIndex**: Removes without retrieving value - O(1) for last index, O(n) otherwise

### Unittests
 - PopFromBeginning : verify popping at index 0 retrieves first element and shifts all
 - PopFromMiddle : verify popping from middle index retrieves correct element and shifts remaining
 - PopFromEnd : verify popping at last index (elementCount-1) retrieves last element
 - ReturnsTrueOnSuccess : verify method returns TRUE when pop succeeds
 - ReturnsFalseOnNegativeIndex : verify FALSE returned for negative index
 - ReturnsFalseOnIndexOutOfBounds : verify FALSE returned when index >= elementCount
 - ReturnsFalseOnEmptyBuffer : verify FALSE returned when buffer is empty (elementCount = 0)
 - WrongElementSize : verify FALSE returned when element size doesn't match
 - EmptyElement : verify behavior when element.diSize is 0 (discard mode)
 - ShiftsElementsCorrectly : verify all elements after index shift left by one position
 - ClearsLastPosition : verify the last position is cleared to zero after shift
 - DecrementsElementCount : verify elementCount decreases by 1 after pop
 - ConsecutivePops : verify multiple consecutive PopAtIndex calls maintain correct state
 - PopAllElements : verify can pop all elements sequentially using index 0
 - ElementOrderPreserved : verify element order is preserved after pop (except removed element)
 - PopAtIndexEquivalentToPopLeft : verify PopAtIndex(0) behaves same as PopLeft
 - PopAtIndexEquivalentToPopRight : verify PopAtIndex(elementCount-1) behaves same as PopRight
*)
PopAtIndex := FALSE;
// Check index bounds, cannot pop what is not filled in
IF index < bufferConfiguration.bufferBoundLower OR index >= bufferConfiguration.bufferBoundLower + bufferMetadata.elementCount THEN
	Trace.Error(__POUNAME(), CONCAT('Pop attempt at invalid index ', TO_STRING(index)));
	RETURN;
END_IF

// Check if buffer is empty
IF isEmpty THEN
	Trace.Error(__POUNAME(), 'Pop attempt on empty buffer');
	RETURN;
END_IF

// rebasedIndex necessary if LL <> 0
rebasedIndex := index - bufferConfiguration.bufferBoundLower;
// TRUE: passed type is not checked, element is discarded and not returned
IF NOT popDiscard THEN
	// Check element size if copy is requested (element.diSize > 0)
	IF element.diSize <> bufferConfiguration.elementSize THEN
		Trace.Error(__POUNAME(), CONCAT('Element size mismatch: expected ', CONCAT(TO_STRING(bufferConfiguration.elementSize), CONCAT(', got ', TO_STRING(element.diSize)))));
		RETURN;
	END_IF

	offset	 := rebasedIndex * bufferConfiguration.elementSize;
	destAddr := element.pValue;
	srcAddr	 := ADR(pBuffer.pValue[offset]);
	nBytes	 := TO_UDINT(element.diSize);
	memcpy(destAddr, srcAddr, nBytes);
END_IF

// Calculate how many elements need to be shifted
elementsToShift := bufferMetadata.elementCount - rebasedIndex - 1;
// Shift elements after the index one position to the left (if any)
IF elementsToShift > 0 THEN
	offset	 := rebasedIndex * bufferConfiguration.elementSize;
	destAddr := ADR(pBuffer.pValue[offset]);								   // destination: current index
	srcAddr	 := ADR(pBuffer.pValue[offset + bufferConfiguration.elementSize]); // source: next index
	nBytes	 := TO_UDINT(elementsToShift * bufferConfiguration.elementSize);
	MEMMOVE(destAddr, srcAddr, nBytes);
END_IF

// Delete last element data 
DeleteAtIndex(bufferMetadata.elementCount + bufferConfiguration.bufferBoundLower - 1);

// Update internal element counters 
CountDecrement();
PopAtIndex := TRUE;
END_METHOD

// Removes and retrieves the first element from the buffer (FIFO/queue operation)
METHOD PopLeft : BOOL
VAR_INPUT
	element	   : ANY;			// Variable to receive the popped element
	popDiscard : BOOL := FALSE; // When TRUE, element is removed but not copied (type checking skipped)
END_VAR

VAR
	offset	 : DINT;
	destAddr : PVOID;
	srcAddr	 : PVOID;
	nBytes	 : UDINT;
END_VAR

(*
## Detailed Description

Removes the first element from the left side of the buffer and optionally copies it to
the provided element parameter. This implements a standard FIFO (First-In-First-Out)
queue operation where elements are dequeued from the front.

The `popDiscard` parameter controls whether the removed element is copied to the output
parameter or simply discarded. This is useful for circular buffer scenarios where you need
to remove elements to make space without retrieving their values.

### Operation Sequence

**When popDiscard = FALSE (default - retrieve element):**
1. Validates that the buffer contains at least one element
2. Validates that element size matches the buffer's configured element size
3. Copies the first element to the output parameter
4. Shifts all remaining elements one position to the left
5. Clears the last position (now empty after the shift)
6. Decrements the element count

**When popDiscard = TRUE (discard element):**
1. Validates that the buffer contains at least one element
2. **Skips element size validation** (type checking bypassed)
3. **Skips copying element** to output parameter
4. Shifts all remaining elements one position to the left
5. Clears the last position (now empty after the shift)
6. Decrements the element count

### Parameters
- **element**: Variable to receive the popped element
  - When popDiscard=FALSE: Must match buffer's element size, receives the popped value
  - When popDiscard=TRUE: Can be any type/size, value is not copied (ignored)
- **popDiscard**: Controls whether to copy element or discard it
  - **FALSE (default)**: Element is validated and copied to output parameter
  - **TRUE**: Element validation is skipped, value is discarded (not copied)
  - Use TRUE for circular buffer overwrite scenarios where you don't need the old value

### Key Features
- **FIFO behavior**: Elements are removed in the order they were added (when combined with PushRight)
- **Optional discard mode**: Can remove element without retrieving it (popDiscard=TRUE)
- **Automatic shifting**: Maintains contiguous element storage after removal
- **Size validation**: Ensures the output element size matches buffer element size (when popDiscard=FALSE)
- **Type safety bypass**: popDiscard=TRUE skips type checking for performance in discard scenarios
- **Safe empty check**: Returns FALSE and logs error if buffer is empty

### Usage Example
```iecst
VAR
    queue : AnyBuffer(pBuffer := myBuffer, bufferBoundLower := 0, bufferBoundUpper := 9, isBufferPersistent := FALSE);
    value : DINT;
    discardBuffer : BYTE;  // Can be any type when using popDiscard=TRUE
    success : BOOL;
END_VAR

// Standard: Pop and retrieve the first element
success := queue.PopLeft(value, FALSE);  // or just queue.PopLeft(value)
IF success THEN
    // Process the retrieved value
END_IF

// Discard mode: Pop without retrieving (e.g., circular buffer overwrite)
success := queue.PopLeft(discardBuffer, TRUE);  // Element removed, value not copied
// OR with temporary pointer-based buffer:
pTemp := __NEW(BYTE, elementSize);
success := queue.PopLeft(pTemp^, TRUE);  // Element removed, discarded to temp buffer
__DELETE(pTemp);
```

### Performance Considerations
- **Time complexity**: O(n) due to element shifting (n = elementCount)
- **Memory operations**: Uses MEMMOVE for efficient bulk memory shifting
- **popDiscard=TRUE**: Slightly faster than popDiscard=FALSE (skips size check and memcpy)
- For frequent left-side operations, consider if a circular buffer would be more efficient

### Return Value
- **TRUE**: Element was successfully popped (and copied if popDiscard=FALSE)
- **FALSE**: Pop operation failed (see error conditions)

### Error Conditions
- Returns FALSE and logs error if buffer is empty (elementCount <= 0)
- Returns FALSE and logs error if element size doesn't match buffer element size **when popDiscard=FALSE**
- When popDiscard=TRUE, element size validation is skipped (no error for size mismatch)

### Dependencies
- Calls DeleteAtIndex to decrement element count and clear the vacated position
- Uses memcpy for element retrieval
- Uses MEMMOVE for shifting elements (handles overlapping memory correctly)
- Uses Trace for error logging

### Unittests
 - RetrievesFirstElement : verify the first element value is copied to output element when popDiscard=FALSE
 - ShiftsElements : verify all elements shift left by one position after pop
 - ClearsLastElement : verify the last position is cleared to zero after shift
 - DecrementsElementCount : verify elementCount decreases by 1 after pop
 - ReturnsTrueOnSuccess : verify method returns TRUE when pop succeeds
 - WrongSize : verify FALSE returned when element size differs from buffer element size (popDiscard=FALSE)
 - EmptyElement : verify behavior when element.diSize is 0 (discard mode, shift only)
 - PopFromEmptyBuffer : verify behavior when buffer has no elements (elementCount = 0)
 - PopSingleElement : verify popping when buffer contains exactly one element
 - ConsecutivePops : verify multiple sequential pops maintain correct order and state
 - PopAfterPushLeft : verify LIFO behavior with PushLeft and PopLeft
 - PopAfterPushRight : verify FIFO behavior with PushRight and PopLeft
 - PopUntilEmpty : verify popping all elements until buffer is empty
 - ElementOrderPreserved : verify remaining elements shift correctly and maintain relative order
 - PopDiscardTrue : verify element is removed but not copied when popDiscard=TRUE
 - PopDiscardTrueSkipsTypeCheck : verify no error when element size is wrong and popDiscard=TRUE
 - PopDiscardTrueShiftsElements : verify elements still shift correctly when popDiscard=TRUE
 - PopDiscardTrueDecrementsCount : verify elementCount decreases when popDiscard=TRUE
 - PopDiscardFalseRetrievesValue : verify element value is copied when popDiscard=FALSE (default)
 - PopDiscardFalseValidatesType : verify type checking occurs when popDiscard=FALSE
 - PopDiscardWithWrongTypeSucceeds : verify PopLeft with wrong type succeeds when popDiscard=TRUE
 - PopDiscardReturnsTrueOnSuccess : verify method returns TRUE when popDiscard=TRUE succeeds
*)
PopLeft := FALSE;
// Check if buffer has elements to pop
IF bufferMetadata.elementCount <= 0 THEN
	Trace.Error(__POUNAME(), 'Cannot pop from empty buffer');
	RETURN;
END_IF

// TRUE: passed type is not checked, element is discarded and not returned
IF NOT popDiscard THEN
	// Check element size if copy is requested (element.diSize > 0)
	IF element.diSize <> bufferConfiguration.elementSize THEN
		Trace.Error(__POUNAME(), CONCAT('Element size mismatch: expected ', CONCAT(TO_STRING(bufferConfiguration.elementSize), CONCAT(', got ', TO_STRING(element.diSize)))));
		RETURN;
	END_IF

	destAddr := element.pValue;
	srcAddr	 := pBuffer.pValue;
	nBytes	 := TO_UDINT(element.diSize);
	memcpy(destAddr, srcAddr, nBytes);
END_IF

// Shift elements to the left
offset	 := bufferConfiguration.elementSize;
destAddr := pBuffer.pValue;
srcAddr	 := ADR(pBuffer.pValue[offset]);
nBytes	 := TO_UDINT((bufferMetadata.elementCount - 1) * bufferConfiguration.elementSize);
MEMMOVE(destAddr, srcAddr, nBytes);

// Delete last element data 
DeleteAtIndex(bufferConfiguration.bufferBoundLower + bufferMetadata.elementCount - 1);

// Update internal element counters 
CountDecrement();
PopLeft := TRUE;
END_METHOD

// Removes and retrieves the last element from the buffer (stack pop operation)
METHOD PopRight : BOOL
VAR_INPUT
	element	   : ANY;			// Variable to receive the popped element
	popDiscard : BOOL := FALSE; // When TRUE, element is removed but not copied (type checking skipped)
END_VAR

VAR
	offset	 : DINT;
	destAddr : PVOID;
	srcAddr	 : PVOID;
	nBytes	 : UDINT;
END_VAR

(*
## Detailed Description

Removes the last element from the right side (back) of the buffer and optionally copies it to
the provided element parameter. This implements a standard stack pop operation where elements
are removed from the back, which can be combined with PushRight for LIFO (Last-In-First-Out)
behavior.

The `popDiscard` parameter controls whether the removed element is copied to the output
parameter or simply discarded. This is useful for circular buffer scenarios where you need
to remove elements to make space without retrieving their values.

### Operation Sequence

